ABB RAPID module: etna.mod

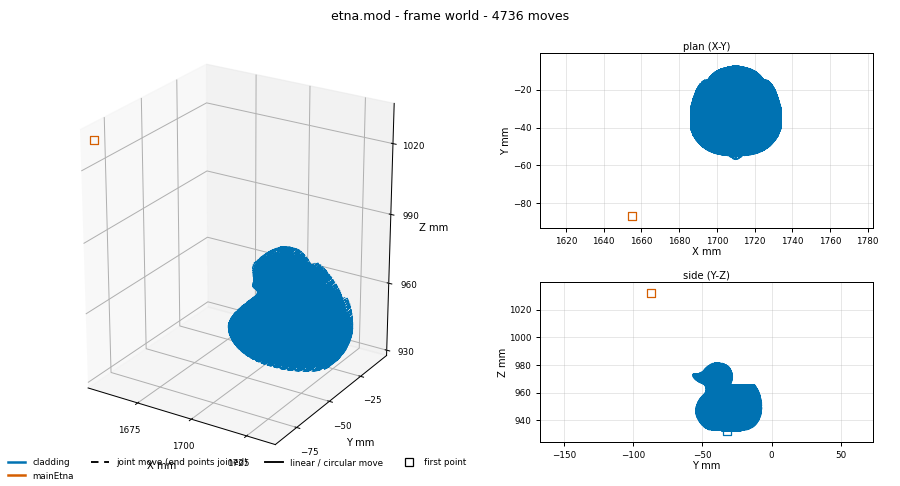
[picture p0: tool path of etna.mod in frame world, 4736 of 4736 moves have a stored position in this frame; points joined in program order, loops and branches not executed]
MODULE Etna

    PERS tooldata toolEtna:=[TRUE,[[530.0,46.8,126.6],[0.707107,0.000000,0.707107,0.000000]],[20,[70,30,123.5],[0,0,1,0],1,0,1]];
    PERS wobjdata wobjEtna:=[FALSE,TRUE,"",[[1655.0,-87.0,932.0],[1.000000,0.000000,0.000000,0.000000]],[[0,0,0],[1,0,0,0]]];

    VAR triggdata laserON;
    VAR triggdata laserOFF;

    CONST speeddata vl:=[8,500,5000,1000];


    CONST robtarget T0:=[[45.230797,54.660942,0.249511],[1.000000,0.000000,0.000000,0.000000],[0,0,-1,0],[9E+09,9E+09,9E+09,9E+09,9E+09,9E+09]];
    CONST robtarget T1:=[[45.230797,61.238206,0.249511],[1.000000,0.000000,0.000000,0.000000],[0,0,-1,0],[9E+09,9E+09,9E+09,9E+09,9E+09,9E+09]];
    CONST robtarget T2:=[[45.230797,54.660942,0.249511],[1.000000,0.000000,0.000000,0.000000],[0,0,-1,0],[9E+09,9E+09,9E+09,9E+09,9E+09,9E+09]];
    CONST robtarget T3:=[[45.230797,61.238206,0.249511],[1.000000,0.000000,0.000000,0.000000],[0,0,-1,0],[9E+09,9E+09,9E+09,9E+09,9E+09,9E+09]];
    CONST robtarget T4:=[[46.730803,63.450242,0.249511],[1.000000,0.000000,0.000000,0.000000],[0,0,-1,0],[9E+09,9E+09,9E+09,9E+09,9E+09,9E+09]];
    CONST robtarget T5:=[[46.730803,53.147305,0.249511],[1.000000,0.000000,0.000000,0.000000],[0,0,-1,0],[9E+09,9E+09,9E+09,9E+09,9E+09,9E+09]];
    CONST robtarget T6:=[[48.230809,51.823648,0.249511],[1.000000,0.000000,0.000000,0.000000],[0,0,-1,0],[9E+09,9E+09,9E+09,9E+09,9E+09,9E+09]];
    CONST robtarget T7:=[[48.230809,64.177413,0.249511],[1.000000,0.000000,0.000000,0.000000],[0,0,-1,0],[9E+09,9E+09,9E+09,9E+09,9E+09,9E+09]];
    CONST robtarget T8:=[[49.730815,64.861657,0.249511],[1.000000,0.000000,0.000000,0.000000],[0,0,-1,0],[9E+09,9E+09,9E+09,9E+09,9E+09,9E+09]];
    CONST robtarget T9:=[[49.730815,50.871953,0.249511],[1.000000,0.000000,0.000000,0.000000],[0,0,-1,0],[9E+09,9E+09,9E+09,9E+09,9E+09,9E+09]];
    CONST robtarget T10:=[[51.230821,50.942602,0.249511],[1.000000,0.000000,0.000000,0.000000],[0,0,-1,0],[9E+09,9E+09,9E+09,9E+09,9E+09,9E+09]];
    CONST robtarget T11:=[[51.230821,64.963902,0.249511],[1.000000,0.000000,0.000000,0.000000],[0,0,-1,0],[9E+09,9E+09,9E+09,9E+09,9E+09,9E+09]];
    CONST robtarget T12:=[[52.730827,64.937092,0.249511],[1.000000,0.000000,0.000000,0.000000],[0,0,-1,0],[9E+09,9E+09,9E+09,9E+09,9E+09,9E+09]];
    CONST robtarget T13:=[[52.730827,51.126270,0.249511],[1.000000,0.000000,0.000000,0.000000],[0,0,-1,0],[9E+09,9E+09,9E+09,9E+09,9E+09,9E+09]];
    CONST robtarget T14:=[[54.230833,51.704495,0.249511],[1.000000,0.000000,0.000000,0.000000],[0,0,-1,0],[9E+09,9E+09,9E+09,9E+09,9E+09,9E+09]];
    CONST robtarget T15:=[[54.230833,64.614973,0.249511],[1.000000,0.000000,0.000000,0.000000],[0,0,-1,0],[9E+09,9E+09,9E+09,9E+09,9E+09,9E+09]];
    CONST robtarget T16:=[[55.730839,64.604426,0.249511],[1.000000,0.000000,0.000000,0.000000],[0,0,-1,0],[9E+09,9E+09,9E+09,9E+09,9E+09,9E+09]];
    CONST robtarget T17:=[[55.730839,51.719275,0.249511],[1.000000,0.000000,0.000000,0.000000],[0,0,-1,0],[9E+09,9E+09,9E+09,9E+09,9E+09,9E+09]];
    CONST robtarget T18:=[[57.230845,51.141050,0.249511],[1.000000,0.000000,0.000000,0.000000],[0,0,-1,0],[9E+09,9E+09,9E+09,9E+09,9E+09,9E+09]];
    CONST robtarget T19:=[[57.230845,64.921597,0.249511],[1.000000,0.000000,0.000000,0.000000],[0,0,-1,0],[9E+09,9E+09,9E+09,9E+09,9E+09,9E+09]];
    CONST robtarget T20:=[[58.730851,64.951383,0.249511],[1.000000,0.000000,0.000000,0.000000],[0,0,-1,0],[9E+09,9E+09,9E+09,9E+09,9E+09,9E+09]];
    CONST robtarget T21:=[[58.730851,50.944648,0.249511],[1.000000,0.000000,0.000000,0.000000],[0,0,-1,0],[9E+09,9E+09,9E+09,9E+09,9E+09,9E+09]];
    CONST robtarget T22:=[[60.230857,50.873711,0.249511],[1.000000,0.000000,0.000000,0.000000],[0,0,-1,0],[9E+09,9E+09,9E+09,9E+09,9E+09,9E+09]];
    CONST robtarget T23:=[[60.230857,64.864853,0.249511],[1.000000,0.000000,0.000000,0.000000],[0,0,-1,0],[9E+09,9E+09,9E+09,9E+09,9E+09,9E+09]];
    CONST robtarget T24:=[[61.730863,64.173309,0.249511],[1.000000,0.000000,0.000000,0.000000],[0,0,-1,0],[9E+09,9E+09,9E+09,9E+09,9E+09,9E+09]];
    CONST robtarget T25:=[[61.730863,51.793503,0.249511],[1.000000,0.000000,0.000000,0.000000],[0,0,-1,0],[9E+09,9E+09,9E+09,9E+09,9E+09,9E+09]];
    CONST robtarget T26:=[[63.230869,53.117219,0.249511],[1.000000,0.000000,0.000000,0.000000],[0,0,-1,0],[9E+09,9E+09,9E+09,9E+09,9E+09,9E+09]];
    CONST robtarget T27:=[[63.230869,63.436121,0.249511],[1.000000,0.000000,0.000000,0.000000],[0,0,-1,0],[9E+09,9E+09,9E+09,9E+09,9E+09,9E+09]];
    CONST robtarget T28:=[[64.730875,61.202460,0.249511],[1.000000,0.000000,0.000000,0.000000],[0,0,-1,0],[9E+09,9E+09,9E+09,9E+09,9E+09,9E+09]];
    CONST robtarget T29:=[[64.730875,54.600120,0.249511],[1.000000,0.000000,0.000000,0.000000],[0,0,-1,0],[9E+09,9E+09,9E+09,9E+09,9E+09,9E+09]];
    CONST robtarget T30:=[[69.247273,52.344904,0.749521],[1.000000,0.000000,0.000000,0.000000],[0,0,-1,0],[9E+09,9E+09,9E+09,9E+09,9E+09,9E+09]];
    CONST robtarget T31:=[[69.247273,59.666876,0.749521],[1.000000,0.000000,0.000000,0.000000],[0,0,-1,0],[9E+09,9E+09,9E+09,9E+09,9E+09,9E+09]];
    CONST robtarget T32:=[[69.247273,52.344904,0.749521],[1.000000,0.000000,0.000000,0.000000],[0,0,-1,0],[9E+09,9E+09,9E+09,9E+09,9E+09,9E+09]];
    CONST robtarget T33:=[[69.247273,59.666876,0.749521],[1.000000,0.000000,0.000000,0.000000],[0,0,-1,0],[9E+09,9E+09,9E+09,9E+09,9E+09,9E+09]];
    CONST robtarget T34:=[[67.747267,63.988813,0.749521],[1.000000,0.000000,0.000000,0.000000],[0,0,-1,0],[9E+09,9E+09,9E+09,9E+09,9E+09,9E+09]];
    CONST robtarget T35:=[[67.747267,49.645310,0.749521],[1.000000,0.000000,0.000000,0.000000],[0,0,-1,0],[9E+09,9E+09,9E+09,9E+09,9E+09,9E+09]];
    CONST robtarget T36:=[[66.247261,47.604168,0.749521],[1.000000,0.000000,0.000000,0.000000],[0,0,-1,0],[9E+09,9E+09,9E+09,9E+09,9E+09,9E+09]];
    CONST robtarget T37:=[[66.247261,65.568560,0.749521],[1.000000,0.000000,0.000000,0.000000],[0,0,-1,0],[9E+09,9E+09,9E+09,9E+09,9E+09,9E+09]];
    CONST robtarget T38:=[[64.747255,66.220066,0.749521],[1.000000,0.000000,0.000000,0.000000],[0,0,-1,0],[9E+09,9E+09,9E+09,9E+09,9E+09,9E+09]];
    CONST robtarget T39:=[[64.747255,46.247530,0.749521],[1.000000,0.000000,0.000000,0.000000],[0,0,-1,0],[9E+09,9E+09,9E+09,9E+09,9E+09,9E+09]];
    CONST robtarget T40:=[[63.247249,45.205197,0.749521],[1.000000,0.000000,0.000000,0.000000],[0,0,-1,0],[9E+09,9E+09,9E+09,9E+09,9E+09,9E+09]];
    CONST robtarget T41:=[[63.247249,66.893237,0.749521],[1.000000,0.000000,0.000000,0.000000],[0,0,-1,0],[9E+09,9E+09,9E+09,9E+09,9E+09,9E+09]];
    CONST robtarget T42:=[[61.747243,67.230044,0.749521],[1.000000,0.000000,0.000000,0.000000],[0,0,-1,0],[9E+09,9E+09,9E+09,9E+09,9E+09,9E+09]];
    CONST robtarget T43:=[[61.747243,44.353778,0.749521],[1.000000,0.000000,0.000000,0.000000],[0,0,-1,0],[9E+09,9E+09,9E+09,9E+09,9E+09,9E+09]];
    CONST robtarget T44:=[[60.247237,43.858747,0.749521],[1.000000,0.000000,0.000000,0.000000],[0,0,-1,0],[9E+09,9E+09,9E+09,9E+09,9E+09,9E+09]];
    CONST robtarget T45:=[[60.247237,67.502036,0.749521],[1.000000,0.000000,0.000000,0.000000],[0,0,-1,0],[9E+09,9E+09,9E+09,9E+09,9E+09,9E+09]];
    CONST robtarget T46:=[[58.747231,67.649975,0.749521],[1.000000,0.000000,0.000000,0.000000],[0,0,-1,0],[9E+09,9E+09,9E+09,9E+09,9E+09,9E+09]];
    CONST robtarget T47:=[[58.747231,43.776283,0.749521],[1.000000,0.000000,0.000000,0.000000],[0,0,-1,0],[9E+09,9E+09,9E+09,9E+09,9E+09,9E+09]];
    CONST robtarget T48:=[[57.247225,43.725602,0.749521],[1.000000,0.000000,0.000000,0.000000],[0,0,-1,0],[9E+09,9E+09,9E+09,9E+09,9E+09,9E+09]];
    CONST robtarget T49:=[[57.247225,67.674292,0.749521],[1.000000,0.000000,0.000000,0.000000],[0,0,-1,0],[9E+09,9E+09,9E+09,9E+09,9E+09,9E+09]];
    CONST robtarget T50:=[[55.747219,67.566917,0.749521],[1.000000,0.000000,0.000000,0.000000],[0,0,-1,0],[9E+09,9E+09,9E+09,9E+09,9E+09,9E+09]];
    CONST robtarget T51:=[[55.747219,43.852921,0.749521],[1.000000,0.000000,0.000000,0.000000],[0,0,-1,0],[9E+09,9E+09,9E+09,9E+09,9E+09,9E+09]];
    CONST robtarget T52:=[[54.247213,43.852451,0.749521],[1.000000,0.000000,0.000000,0.000000],[0,0,-1,0],[9E+09,9E+09,9E+09,9E+09,9E+09,9E+09]];
    CONST robtarget T53:=[[54.247213,67.567771,0.749521],[1.000000,0.000000,0.000000,0.000000],[0,0,-1,0],[9E+09,9E+09,9E+09,9E+09,9E+09,9E+09]];
    CONST robtarget T54:=[[52.747207,67.674435,0.749521],[1.000000,0.000000,0.000000,0.000000],[0,0,-1,0],[9E+09,9E+09,9E+09,9E+09,9E+09,9E+09]];
    CONST robtarget T55:=[[52.747207,43.725093,0.749521],[1.000000,0.000000,0.000000,0.000000],[0,0,-1,0],[9E+09,9E+09,9E+09,9E+09,9E+09,9E+09]];
    CONST robtarget T56:=[[51.247201,43.776532,0.749521],[1.000000,0.000000,0.000000,0.000000],[0,0,-1,0],[9E+09,9E+09,9E+09,9E+09,9E+09,9E+09]];
    CONST robtarget T57:=[[51.247201,67.650171,0.749521],[1.000000,0.000000,0.000000,0.000000],[0,0,-1,0],[9E+09,9E+09,9E+09,9E+09,9E+09,9E+09]];
    CONST robtarget T58:=[[49.747195,67.501890,0.749521],[1.000000,0.000000,0.000000,0.000000],[0,0,-1,0],[9E+09,9E+09,9E+09,9E+09,9E+09,9E+09]];
    CONST robtarget T59:=[[49.747195,43.860589,0.749521],[1.000000,0.000000,0.000000,0.000000],[0,0,-1,0],[9E+09,9E+09,9E+09,9E+09,9E+09,9E+09]];
    CONST robtarget T60:=[[48.247189,44.355622,0.749521],[1.000000,0.000000,0.000000,0.000000],[0,0,-1,0],[9E+09,9E+09,9E+09,9E+09,9E+09,9E+09]];
    CONST robtarget T61:=[[48.247189,67.230329,0.749521],[1.000000,0.000000,0.000000,0.000000],[0,0,-1,0],[9E+09,9E+09,9E+09,9E+09,9E+09,9E+09]];
    CONST robtarget T62:=[[46.747183,66.892498,0.749521],[1.000000,0.000000,0.000000,0.000000],[0,0,-1,0],[9E+09,9E+09,9E+09,9E+09,9E+09,9E+09]];
    CONST robtarget T63:=[[46.747183,45.207884,0.749521],[1.000000,0.000000,0.000000,0.000000],[0,0,-1,0],[9E+09,9E+09,9E+09,9E+09,9E+09,9E+09]];
    CONST robtarget T64:=[[45.247177,46.252109,0.749521],[1.000000,0.000000,0.000000,0.000000],[0,0,-1,0],[9E+09,9E+09,9E+09,9E+09,9E+09,9E+09]];
    CONST robtarget T65:=[[45.247177,66.220428,0.749521],[1.000000,0.000000,0.000000,0.000000],[0,0,-1,0],[9E+09,9E+09,9E+09,9E+09,9E+09,9E+09]];
    CONST robtarget T66:=[[43.747171,65.569397,0.749521],[1.000000,0.000000,0.000000,0.000000],[0,0,-1,0],[9E+09,9E+09,9E+09,9E+09,9E+09,9E+09]];
    CONST robtarget T67:=[[43.747171,47.613223,0.749521],[1.000000,0.000000,0.000000,0.000000],[0,0,-1,0],[9E+09,9E+09,9E+09,9E+09,9E+09,9E+09]];
    CONST robtarget T68:=[[42.247165,49.652254,0.749521],[1.000000,0.000000,0.000000,0.000000],[0,0,-1,0],[9E+09,9E+09,9E+09,9E+09,9E+09,9E+09]];
    CONST robtarget T69:=[[42.247165,63.997482,0.749521],[1.000000,0.000000,0.000000,0.000000],[0,0,-1,0],[9E+09,9E+09,9E+09,9E+09,9E+09,9E+09]];
    CONST robtarget T70:=[[40.747159,59.721737,0.749521],[1.000000,0.000000,0.000000,0.000000],[0,0,-1,0],[9E+09,9E+09,9E+09,9E+09,9E+09,9E+09]];
    CONST robtarget T71:=[[40.747159,52.382179,0.749521],[1.000000,0.000000,0.000000,0.000000],[0,0,-1,0],[9E+09,9E+09,9E+09,9E+09,9E+09,9E+09]];
    CONST robtarget T72:=[[38.499544,50.308177,1.249531],[1.000000,0.000000,0.000000,0.000000],[0,0,-1,0],[9E+09,9E+09,9E+09,9E+09,9E+09,9E+09]];
    CONST robtarget T73:=[[38.499544,60.298450,1.249531],[1.000000,0.000000,0.000000,0.000000],[0,0,-1,0],[9E+09,9E+09,9E+09,9E+09,9E+09,9E+09]];
    CONST robtarget T74:=[[38.499544,50.308177,1.249531],[1.000000,0.000000,0.000000,0.000000],[0,0,-1,0],[9E+09,9E+09,9E+09,9E+09,9E+09,9E+09]];
    CONST robtarget T75:=[[38.499544,60.298450,1.249531],[1.000000,0.000000,0.000000,0.000000],[0,0,-1,0],[9E+09,9E+09,9E+09,9E+09,9E+09,9E+09]];
    CONST robtarget T76:=[[39.999550,64.489479,1.249531],[1.000000,0.000000,0.000000,0.000000],[0,0,-1,0],[9E+09,9E+09,9E+09,9E+09,9E+09,9E+09]];
    CONST robtarget T77:=[[39.999550,47.499380,1.249531],[1.000000,0.000000,0.000000,0.000000],[0,0,-1,0],[9E+09,9E+09,9E+09,9E+09,9E+09,9E+09]];
    CONST robtarget T78:=[[41.499556,46.077025,1.249531],[1.000000,0.000000,0.000000,0.000000],[0,0,-1,0],[9E+09,9E+09,9E+09,9E+09,9E+09,9E+09]];
    CONST robtarget T79:=[[41.499556,66.064956,1.249531],[1.000000,0.000000,0.000000,0.000000],[0,0,-1,0],[9E+09,9E+09,9E+09,9E+09,9E+09,9E+09]];
    CONST robtarget T80:=[[42.999562,67.172158,1.249531],[1.000000,0.000000,0.000000,0.000000],[0,0,-1,0],[9E+09,9E+09,9E+09,9E+09,9E+09,9E+09]];
    CONST robtarget T81:=[[42.999562,44.769816,1.249531],[1.000000,0.000000,0.000000,0.000000],[0,0,-1,0],[9E+09,9E+09,9E+09,9E+09,9E+09,9E+09]];
    CONST robtarget T82:=[[44.499568,44.074901,1.249531],[1.000000,0.000000,0.000000,0.000000],[0,0,-1,0],[9E+09,9E+09,9E+09,9E+09,9E+09,9E+09]];
    CONST robtarget T83:=[[44.499568,68.035223,1.249531],[1.000000,0.000000,0.000000,0.000000],[0,0,-1,0],[9E+09,9E+09,9E+09,9E+09,9E+09,9E+09]];
    CONST robtarget T84:=[[45.999574,68.487089,1.249531],[1.000000,0.000000,0.000000,0.000000],[0,0,-1,0],[9E+09,9E+09,9E+09,9E+09,9E+09,9E+09]];
    CONST robtarget T85:=[[45.999574,43.291383,1.249531],[1.000000,0.000000,0.000000,0.000000],[0,0,-1,0],[9E+09,9E+09,9E+09,9E+09,9E+09,9E+09]];
    CONST robtarget T86:=[[47.499580,42.569706,1.249531],[1.000000,0.000000,0.000000,0.000000],[0,0,-1,0],[9E+09,9E+09,9E+09,9E+09,9E+09,9E+09]];
    CONST robtarget T87:=[[47.499580,68.938955,1.249531],[1.000000,0.000000,0.000000,0.000000],[0,0,-1,0],[9E+09,9E+09,9E+09,9E+09,9E+09,9E+09]];
    CONST robtarget T88:=[[48.999586,69.156373,1.249531],[1.000000,0.000000,0.000000,0.000000],[0,0,-1,0],[9E+09,9E+09,9E+09,9E+09,9E+09,9E+09]];
    CONST robtarget T89:=[[48.999586,42.028761,1.249531],[1.000000,0.000000,0.000000,0.000000],[0,0,-1,0],[9E+09,9E+09,9E+09,9E+09,9E+09,9E+09]];
    CONST robtarget T90:=[[50.499592,41.629502,1.249531],[1.000000,0.000000,0.000000,0.000000],[0,0,-1,0],[9E+09,9E+09,9E+09,9E+09,9E+09,9E+09]];
    CONST robtarget T91:=[[50.499592,69.313504,1.249531],[1.000000,0.000000,0.000000,0.000000],[0,0,-1,0],[9E+09,9E+09,9E+09,9E+09,9E+09,9E+09]];
    CONST robtarget T92:=[[51.999598,69.380595,1.249531],[1.000000,0.000000,0.000000,0.000000],[0,0,-1,0],[9E+09,9E+09,9E+09,9E+09,9E+09,9E+09]];
    CONST robtarget T93:=[[51.999598,41.543714,1.249531],[1.000000,0.000000,0.000000,0.000000],[0,0,-1,0],[9E+09,9E+09,9E+09,9E+09,9E+09,9E+09]];
    CONST robtarget T94:=[[53.499604,41.519114,1.249531],[1.000000,0.000000,0.000000,0.000000],[0,0,-1,0],[9E+09,9E+09,9E+09,9E+09,9E+09,9E+09]];
    CONST robtarget T95:=[[53.499604,69.370940,1.249531],[1.000000,0.000000,0.000000,0.000000],[0,0,-1,0],[9E+09,9E+09,9E+09,9E+09,9E+09,9E+09]];
    CONST robtarget T96:=[[54.999610,69.325352,1.249531],[1.000000,0.000000,0.000000,0.000000],[0,0,-1,0],[9E+09,9E+09,9E+09,9E+09,9E+09,9E+09]];
    CONST robtarget T97:=[[54.999610,41.622696,1.249531],[1.000000,0.000000,0.000000,0.000000],[0,0,-1,0],[9E+09,9E+09,9E+09,9E+09,9E+09,9E+09]];
    CONST robtarget T98:=[[56.499616,41.519131,1.249531],[1.000000,0.000000,0.000000,0.000000],[0,0,-1,0],[9E+09,9E+09,9E+09,9E+09,9E+09,9E+09]];
    CONST robtarget T99:=[[56.499616,69.370908,1.249531],[1.000000,0.000000,0.000000,0.000000],[0,0,-1,0],[9E+09,9E+09,9E+09,9E+09,9E+09,9E+09]];
    CONST robtarget T100:=[[57.999622,69.380616,1.249531],[1.000000,0.000000,0.000000,0.000000],[0,0,-1,0],[9E+09,9E+09,9E+09,9E+09,9E+09,9E+09]];
    CONST robtarget T101:=[[57.999622,41.543669,1.249531],[1.000000,0.000000,0.000000,0.000000],[0,0,-1,0],[9E+09,9E+09,9E+09,9E+09,9E+09,9E+09]];
    CONST robtarget T102:=[[59.499628,41.629457,1.249531],[1.000000,0.000000,0.000000,0.000000],[0,0,-1,0],[9E+09,9E+09,9E+09,9E+09,9E+09,9E+09]];
    CONST robtarget T103:=[[59.499628,69.313582,1.249531],[1.000000,0.000000,0.000000,0.000000],[0,0,-1,0],[9E+09,9E+09,9E+09,9E+09,9E+09,9E+09]];
    CONST robtarget T104:=[[60.999634,69.156474,1.249531],[1.000000,0.000000,0.000000,0.000000],[0,0,-1,0],[9E+09,9E+09,9E+09,9E+09,9E+09,9E+09]];
    CONST robtarget T105:=[[60.999634,42.028474,1.249531],[1.000000,0.000000,0.000000,0.000000],[0,0,-1,0],[9E+09,9E+09,9E+09,9E+09,9E+09,9E+09]];
    CONST robtarget T106:=[[62.499640,42.569419,1.249531],[1.000000,0.000000,0.000000,0.000000],[0,0,-1,0],[9E+09,9E+09,9E+09,9E+09,9E+09,9E+09]];
    CONST robtarget T107:=[[62.499640,68.939194,1.249531],[1.000000,0.000000,0.000000,0.000000],[0,0,-1,0],[9E+09,9E+09,9E+09,9E+09,9E+09,9E+09]];
    CONST robtarget T108:=[[63.999646,68.487328,1.249531],[1.000000,0.000000,0.000000,0.000000],[0,0,-1,0],[9E+09,9E+09,9E+09,9E+09,9E+09,9E+09]];
    CONST robtarget T109:=[[63.999646,43.290925,1.249531],[1.000000,0.000000,0.000000,0.000000],[0,0,-1,0],[9E+09,9E+09,9E+09,9E+09,9E+09,9E+09]];
    CONST robtarget T110:=[[65.499652,44.074529,1.249531],[1.000000,0.000000,0.000000,0.000000],[0,0,-1,0],[9E+09,9E+09,9E+09,9E+09,9E+09,9E+09]];
    CONST robtarget T111:=[[65.499652,68.035462,1.249531],[1.000000,0.000000,0.000000,0.000000],[0,0,-1,0],[9E+09,9E+09,9E+09,9E+09,9E+09,9E+09]];
    CONST robtarget T112:=[[66.999658,67.172468,1.249531],[1.000000,0.000000,0.000000,0.000000],[0,0,-1,0],[9E+09,9E+09,9E+09,9E+09,9E+09,9E+09]];
    CONST robtarget T113:=[[66.999658,44.769447,1.249531],[1.000000,0.000000,0.000000,0.000000],[0,0,-1,0],[9E+09,9E+09,9E+09,9E+09,9E+09,9E+09]];
    CONST robtarget T114:=[[68.499664,46.076202,1.249531],[1.000000,0.000000,0.000000,0.000000],[0,0,-1,0],[9E+09,9E+09,9E+09,9E+09,9E+09,9E+09]];
    CONST robtarget T115:=[[68.499664,66.065017,1.249531],[1.000000,0.000000,0.000000,0.000000],[0,0,-1,0],[9E+09,9E+09,9E+09,9E+09,9E+09,9E+09]];
    CONST robtarget T116:=[[69.999670,64.488299,1.249531],[1.000000,0.000000,0.000000,0.000000],[0,0,-1,0],[9E+09,9E+09,9E+09,9E+09,9E+09,9E+09]];
    CONST robtarget T117:=[[69.999670,47.498673,1.249531],[1.000000,0.000000,0.000000,0.000000],[0,0,-1,0],[9E+09,9E+09,9E+09,9E+09,9E+09,9E+09]];
    CONST robtarget T118:=[[71.499676,50.306050,1.249531],[1.000000,0.000000,0.000000,0.000000],[0,0,-1,0],[9E+09,9E+09,9E+09,9E+09,9E+09,9E+09]];
    CONST robtarget T119:=[[71.499676,60.263678,1.249531],[1.000000,0.000000,0.000000,0.000000],[0,0,-1,0],[9E+09,9E+09,9E+09,9E+09,9E+09,9E+09]];
    CONST robtarget T120:=[[73.000077,49.540950,1.749541],[1.000000,0.000000,0.000000,0.000000],[0,0,-1,0],[9E+09,9E+09,9E+09,9E+09,9E+09,9E+09]];
    CONST robtarget T121:=[[73.000077,58.164737,1.749541],[1.000000,0.000000,0.000000,0.000000],[0,0,-1,0],[9E+09,9E+09,9E+09,9E+09,9E+09,9E+09]];
    CONST robtarget T122:=[[73.000077,49.540950,1.749541],[1.000000,0.000000,0.000000,0.000000],[0,0,-1,0],[9E+09,9E+09,9E+09,9E+09,9E+09,9E+09]];
    CONST robtarget T123:=[[73.000077,58.164737,1.749541],[1.000000,0.000000,0.000000,0.000000],[0,0,-1,0],[9E+09,9E+09,9E+09,9E+09,9E+09,9E+09]];
    CONST robtarget T124:=[[71.500071,63.783623,1.749541],[1.000000,0.000000,0.000000,0.000000],[0,0,-1,0],[9E+09,9E+09,9E+09,9E+09,9E+09,9E+09]];
    CONST robtarget T125:=[[71.500071,46.656280,1.749541],[1.000000,0.000000,0.000000,0.000000],[0,0,-1,0],[9E+09,9E+09,9E+09,9E+09,9E+09,9E+09]];
    CONST robtarget T126:=[[70.000065,45.101701,1.749541],[1.000000,0.000000,0.000000,0.000000],[0,0,-1,0],[9E+09,9E+09,9E+09,9E+09,9E+09,9E+09]];
    CONST robtarget T127:=[[70.000065,66.271272,1.749541],[1.000000,0.000000,0.000000,0.000000],[0,0,-1,0],[9E+09,9E+09,9E+09,9E+09,9E+09,9E+09]];
    CONST robtarget T128:=[[68.500059,67.688442,1.749541],[1.000000,0.000000,0.000000,0.000000],[0,0,-1,0],[9E+09,9E+09,9E+09,9E+09,9E+09,9E+09]];
    CONST robtarget T129:=[[68.500059,44.151934,1.749541],[1.000000,0.000000,0.000000,0.000000],[0,0,-1,0],[9E+09,9E+09,9E+09,9E+09,9E+09,9E+09]];
    CONST robtarget T130:=[[67.000053,43.202167,1.749541],[1.000000,0.000000,0.000000,0.000000],[0,0,-1,0],[9E+09,9E+09,9E+09,9E+09,9E+09,9E+09]];
    CONST robtarget T131:=[[67.000053,68.457961,1.749541],[1.000000,0.000000,0.000000,0.000000],[0,0,-1,0],[9E+09,9E+09,9E+09,9E+09,9E+09,9E+09]];
    CONST robtarget T132:=[[65.500047,69.385771,1.749541],[1.000000,0.000000,0.000000,0.000000],[0,0,-1,0],[9E+09,9E+09,9E+09,9E+09,9E+09,9E+09]];
    CONST robtarget T133:=[[65.500047,42.445663,1.749541],[1.000000,0.000000,0.000000,0.000000],[0,0,-1,0],[9E+09,9E+09,9E+09,9E+09,9E+09,9E+09]];
    CONST robtarget T134:=[[64.000041,41.874691,1.749541],[1.000000,0.000000,0.000000,0.000000],[0,0,-1,0],[9E+09,9E+09,9E+09,9E+09,9E+09,9E+09]];
    CONST robtarget T135:=[[64.000041,69.938803,1.749541],[1.000000,0.000000,0.000000,0.000000],[0,0,-1,0],[9E+09,9E+09,9E+09,9E+09,9E+09,9E+09]];
    CONST robtarget T136:=[[62.500035,70.380115,1.749541],[1.000000,0.000000,0.000000,0.000000],[0,0,-1,0],[9E+09,9E+09,9E+09,9E+09,9E+09,9E+09]];
    CONST robtarget T137:=[[62.500035,41.341429,1.749541],[1.000000,0.000000,0.000000,0.000000],[0,0,-1,0],[9E+09,9E+09,9E+09,9E+09,9E+09,9E+09]];
    CONST robtarget T138:=[[61.000029,40.952491,1.749541],[1.000000,0.000000,0.000000,0.000000],[0,0,-1,0],[9E+09,9E+09,9E+09,9E+09,9E+09,9E+09]];
    CONST robtarget T139:=[[61.000029,70.613365,1.749541],[1.000000,0.000000,0.000000,0.000000],[0,0,-1,0],[9E+09,9E+09,9E+09,9E+09,9E+09,9E+09]];
    CONST robtarget T140:=[[59.500023,70.730845,1.749541],[1.000000,0.000000,0.000000,0.000000],[0,0,-1,0],[9E+09,9E+09,9E+09,9E+09,9E+09,9E+09]];
    CONST robtarget T141:=[[59.500023,40.606692,1.749541],[1.000000,0.000000,0.000000,0.000000],[0,0,-1,0],[9E+09,9E+09,9E+09,9E+09,9E+09,9E+09]];
    CONST robtarget T142:=[[58.000017,40.513780,1.749541],[1.000000,0.000000,0.000000,0.000000],[0,0,-1,0],[9E+09,9E+09,9E+09,9E+09,9E+09,9E+09]];
    CONST robtarget T143:=[[58.000017,70.803110,1.749541],[1.000000,0.000000,0.000000,0.000000],[0,0,-1,0],[9E+09,9E+09,9E+09,9E+09,9E+09,9E+09]];
    CONST robtarget T144:=[[56.500011,70.842486,1.749541],[1.000000,0.000000,0.000000,0.000000],[0,0,-1,0],[9E+09,9E+09,9E+09,9E+09,9E+09,9E+09]];
    CONST robtarget T145:=[[56.500011,40.485362,1.749541],[1.000000,0.000000,0.000000,0.000000],[0,0,-1,0],[9E+09,9E+09,9E+09,9E+09,9E+09,9E+09]];
    CONST robtarget T146:=[[55.000005,40.512783,1.749541],[1.000000,0.000000,0.000000,0.000000],[0,0,-1,0],[9E+09,9E+09,9E+09,9E+09,9E+09,9E+09]];
    CONST robtarget T147:=[[55.000005,70.830121,1.749541],[1.000000,0.000000,0.000000,0.000000],[0,0,-1,0],[9E+09,9E+09,9E+09,9E+09,9E+09,9E+09]];
    CONST robtarget T148:=[[53.499999,70.842488,1.749541],[1.000000,0.000000,0.000000,0.000000],[0,0,-1,0],[9E+09,9E+09,9E+09,9E+09,9E+09,9E+09]];
    CONST robtarget T149:=[[53.499999,40.485362,1.749541],[1.000000,0.000000,0.000000,0.000000],[0,0,-1,0],[9E+09,9E+09,9E+09,9E+09,9E+09,9E+09]];
    CONST robtarget T150:=[[51.999993,40.513780,1.749541],[1.000000,0.000000,0.000000,0.000000],[0,0,-1,0],[9E+09,9E+09,9E+09,9E+09,9E+09,9E+09]];
    CONST robtarget T151:=[[51.999993,70.803110,1.749541],[1.000000,0.000000,0.000000,0.000000],[0,0,-1,0],[9E+09,9E+09,9E+09,9E+09,9E+09,9E+09]];
    CONST robtarget T152:=[[50.499987,70.730845,1.749541],[1.000000,0.000000,0.000000,0.000000],[0,0,-1,0],[9E+09,9E+09,9E+09,9E+09,9E+09,9E+09]];
    CONST robtarget T153:=[[50.499987,40.606692,1.749541],[1.000000,0.000000,0.000000,0.000000],[0,0,-1,0],[9E+09,9E+09,9E+09,9E+09,9E+09,9E+09]];
    CONST robtarget T154:=[[48.999981,40.952493,1.749541],[1.000000,0.000000,0.000000,0.000000],[0,0,-1,0],[9E+09,9E+09,9E+09,9E+09,9E+09,9E+09]];
    CONST robtarget T155:=[[48.999981,70.613365,1.749541],[1.000000,0.000000,0.000000,0.000000],[0,0,-1,0],[9E+09,9E+09,9E+09,9E+09,9E+09,9E+09]];
    CONST robtarget T156:=[[47.499975,70.380114,1.749541],[1.000000,0.000000,0.000000,0.000000],[0,0,-1,0],[9E+09,9E+09,9E+09,9E+09,9E+09,9E+09]];
    CONST robtarget T157:=[[47.499975,41.341430,1.749541],[1.000000,0.000000,0.000000,0.000000],[0,0,-1,0],[9E+09,9E+09,9E+09,9E+09,9E+09,9E+09]];
    CONST robtarget T158:=[[45.999969,41.874694,1.749541],[1.000000,0.000000,0.000000,0.000000],[0,0,-1,0],[9E+09,9E+09,9E+09,9E+09,9E+09,9E+09]];
    CONST robtarget T159:=[[45.999969,69.938801,1.749541],[1.000000,0.000000,0.000000,0.000000],[0,0,-1,0],[9E+09,9E+09,9E+09,9E+09,9E+09,9E+09]];
    CONST robtarget T160:=[[44.499963,69.385768,1.749541],[1.000000,0.000000,0.000000,0.000000],[0,0,-1,0],[9E+09,9E+09,9E+09,9E+09,9E+09,9E+09]];
    CONST robtarget T161:=[[44.499963,42.445669,1.749541],[1.000000,0.000000,0.000000,0.000000],[0,0,-1,0],[9E+09,9E+09,9E+09,9E+09,9E+09,9E+09]];
    CONST robtarget T162:=[[42.999957,43.202177,1.749541],[1.000000,0.000000,0.000000,0.000000],[0,0,-1,0],[9E+09,9E+09,9E+09,9E+09,9E+09,9E+09]];
    CONST robtarget T163:=[[42.999957,68.457958,1.749541],[1.000000,0.000000,0.000000,0.000000],[0,0,-1,0],[9E+09,9E+09,9E+09,9E+09,9E+09,9E+09]];
    CONST robtarget T164:=[[41.499951,67.688441,1.749541],[1.000000,0.000000,0.000000,0.000000],[0,0,-1,0],[9E+09,9E+09,9E+09,9E+09,9E+09,9E+09]];
    CONST robtarget T165:=[[41.499951,44.151941,1.749541],[1.000000,0.000000,0.000000,0.000000],[0,0,-1,0],[9E+09,9E+09,9E+09,9E+09,9E+09,9E+09]];
    CONST robtarget T166:=[[39.999945,45.101704,1.749541],[1.000000,0.000000,0.000000,0.000000],[0,0,-1,0],[9E+09,9E+09,9E+09,9E+09,9E+09,9E+09]];
    CONST robtarget T167:=[[39.999945,66.272627,1.749541],[1.000000,0.000000,0.000000,0.000000],[0,0,-1,0],[9E+09,9E+09,9E+09,9E+09,9E+09,9E+09]];
    CONST robtarget T168:=[[38.499939,63.788624,1.749541],[1.000000,0.000000,0.000000,0.000000],[0,0,-1,0],[9E+09,9E+09,9E+09,9E+09,9E+09,9E+09]];
    CONST robtarget T169:=[[38.499939,46.656285,1.749541],[1.000000,0.000000,0.000000,0.000000],[0,0,-1,0],[9E+09,9E+09,9E+09,9E+09,9E+09,9E+09]];
    CONST robtarget T170:=[[36.999933,49.540961,1.749541],[1.000000,0.000000,0.000000,0.000000],[0,0,-1,0],[9E+09,9E+09,9E+09,9E+09,9E+09,9E+09]];
    CONST robtarget T171:=[[36.999933,58.175696,1.749541],[1.000000,0.000000,0.000000,0.000000],[0,0,-1,0],[9E+09,9E+09,9E+09,9E+09,9E+09,9E+09]];
    CONST robtarget T172:=[[36.250324,48.397228,2.249551],[1.000000,0.000000,0.000000,0.000000],[0,0,-1,0],[9E+09,9E+09,9E+09,9E+09,9E+09,9E+09]];
    CONST robtarget T173:=[[36.250324,59.214847,2.249551],[1.000000,0.000000,0.000000,0.000000],[0,0,-1,0],[9E+09,9E+09,9E+09,9E+09,9E+09,9E+09]];
    CONST robtarget T174:=[[36.250324,48.397228,2.249551],[1.000000,0.000000,0.000000,0.000000],[0,0,-1,0],[9E+09,9E+09,9E+09,9E+09,9E+09,9E+09]];
    CONST robtarget T175:=[[36.250324,59.214847,2.249551],[1.000000,0.000000,0.000000,0.000000],[0,0,-1,0],[9E+09,9E+09,9E+09,9E+09,9E+09,9E+09]];
    CONST robtarget T176:=[[37.750330,64.085193,2.249551],[1.000000,0.000000,0.000000,0.000000],[0,0,-1,0],[9E+09,9E+09,9E+09,9E+09,9E+09,9E+09]];
    CONST robtarget T177:=[[37.750330,45.991942,2.249551],[1.000000,0.000000,0.000000,0.000000],[0,0,-1,0],[9E+09,9E+09,9E+09,9E+09,9E+09,9E+09]];
    CONST robtarget T178:=[[39.250336,44.568903,2.249551],[1.000000,0.000000,0.000000,0.000000],[0,0,-1,0],[9E+09,9E+09,9E+09,9E+09,9E+09,9E+09]];
    CONST robtarget T179:=[[39.250336,66.308930,2.249551],[1.000000,0.000000,0.000000,0.000000],[0,0,-1,0],[9E+09,9E+09,9E+09,9E+09,9E+09,9E+09]];
    CONST robtarget T180:=[[40.750342,67.989973,2.249551],[1.000000,0.000000,0.000000,0.000000],[0,0,-1,0],[9E+09,9E+09,9E+09,9E+09,9E+09,9E+09]];
    CONST robtarget T181:=[[40.750342,43.327424,2.249551],[1.000000,0.000000,0.000000,0.000000],[0,0,-1,0],[9E+09,9E+09,9E+09,9E+09,9E+09,9E+09]];
    CONST robtarget T182:=[[42.250348,42.606898,2.249551],[1.000000,0.000000,0.000000,0.000000],[0,0,-1,0],[9E+09,9E+09,9E+09,9E+09,9E+09,9E+09]];
    CONST robtarget T183:=[[42.250348,69.121905,2.249551],[1.000000,0.000000,0.000000,0.000000],[0,0,-1,0],[9E+09,9E+09,9E+09,9E+09,9E+09,9E+09]];
    CONST robtarget T184:=[[43.750354,70.008448,2.249551],[1.000000,0.000000,0.000000,0.000000],[0,0,-1,0],[9E+09,9E+09,9E+09,9E+09,9E+09,9E+09]];
    CONST robtarget T185:=[[43.750354,41.846430,2.249551],[1.000000,0.000000,0.000000,0.000000],[0,0,-1,0],[9E+09,9E+09,9E+09,9E+09,9E+09,9E+09]];
    CONST robtarget T186:=[[45.250360,41.202387,2.249551],[1.000000,0.000000,0.000000,0.000000],[0,0,-1,0],[9E+09,9E+09,9E+09,9E+09,9E+09,9E+09]];
    CONST robtarget T187:=[[45.250360,70.831245,2.249551],[1.000000,0.000000,0.000000,0.000000],[0,0,-1,0],[9E+09,9E+09,9E+09,9E+09,9E+09,9E+09]];
    CONST robtarget T188:=[[46.750366,71.247041,2.249551],[1.000000,0.000000,0.000000,0.000000],[0,0,-1,0],[9E+09,9E+09,9E+09,9E+09,9E+09,9E+09]];
    CONST robtarget T189:=[[46.750366,40.618606,2.249551],[1.000000,0.000000,0.000000,0.000000],[0,0,-1,0],[9E+09,9E+09,9E+09,9E+09,9E+09,9E+09]];
    CONST robtarget T190:=[[48.250372,40.149877,2.249551],[1.000000,0.000000,0.000000,0.000000],[0,0,-1,0],[9E+09,9E+09,9E+09,9E+09,9E+09,9E+09]];
    CONST robtarget T191:=[[48.250372,71.629090,2.249551],[1.000000,0.000000,0.000000,0.000000],[0,0,-1,0],[9E+09,9E+09,9E+09,9E+09,9E+09,9E+09]];
    CONST robtarget T192:=[[49.750378,71.805464,2.249551],[1.000000,0.000000,0.000000,0.000000],[0,0,-1,0],[9E+09,9E+09,9E+09,9E+09,9E+09,9E+09]];
    CONST robtarget T193:=[[49.750378,39.761399,2.249551],[1.000000,0.000000,0.000000,0.000000],[0,0,-1,0],[9E+09,9E+09,9E+09,9E+09,9E+09,9E+09]];
    CONST robtarget T194:=[[51.250384,39.536943,2.249551],[1.000000,0.000000,0.000000,0.000000],[0,0,-1,0],[9E+09,9E+09,9E+09,9E+09,9E+09,9E+09]];
    CONST robtarget T195:=[[51.250384,71.906931,2.249551],[1.000000,0.000000,0.000000,0.000000],[0,0,-1,0],[9E+09,9E+09,9E+09,9E+09,9E+09,9E+09]];
    CONST robtarget T196:=[[52.750390,71.973450,2.249551],[1.000000,0.000000,0.000000,0.000000],[0,0,-1,0],[9E+09,9E+09,9E+09,9E+09,9E+09,9E+09]];
    CONST robtarget T197:=[[52.750390,39.440952,2.249551],[1.000000,0.000000,0.000000,0.000000],[0,0,-1,0],[9E+09,9E+09,9E+09,9E+09,9E+09,9E+09]];
    CONST robtarget T198:=[[54.250396,39.462104,2.249551],[1.000000,0.000000,0.000000,0.000000],[0,0,-1,0],[9E+09,9E+09,9E+09,9E+09,9E+09,9E+09]];
    CONST robtarget T199:=[[54.250396,72.010261,2.249551],[1.000000,0.000000,0.000000,0.000000],[0,0,-1,0],[9E+09,9E+09,9E+09,9E+09,9E+09,9E+09]];
    CONST robtarget T200:=[[55.750402,72.010251,2.249551],[1.000000,0.000000,0.000000,0.000000],[0,0,-1,0],[9E+09,9E+09,9E+09,9E+09,9E+09,9E+09]];
    CONST robtarget T201:=[[55.750402,39.462091,2.249551],[1.000000,0.000000,0.000000,0.000000],[0,0,-1,0],[9E+09,9E+09,9E+09,9E+09,9E+09,9E+09]];
    CONST robtarget T202:=[[57.250408,39.440997,2.249551],[1.000000,0.000000,0.000000,0.000000],[0,0,-1,0],[9E+09,9E+09,9E+09,9E+09,9E+09,9E+09]];
    CONST robtarget T203:=[[57.250408,71.973400,2.249551],[1.000000,0.000000,0.000000,0.000000],[0,0,-1,0],[9E+09,9E+09,9E+09,9E+09,9E+09,9E+09]];
    CONST robtarget T204:=[[58.750414,71.906869,2.249551],[1.000000,0.000000,0.000000,0.000000],[0,0,-1,0],[9E+09,9E+09,9E+09,9E+09,9E+09,9E+09]];
    CONST robtarget T205:=[[58.750414,39.536995,2.249551],[1.000000,0.000000,0.000000,0.000000],[0,0,-1,0],[9E+09,9E+09,9E+09,9E+09,9E+09,9E+09]];
    CONST robtarget T206:=[[60.250420,39.761602,2.249551],[1.000000,0.000000,0.000000,0.000000],[0,0,-1,0],[9E+09,9E+09,9E+09,9E+09,9E+09,9E+09]];
    CONST robtarget T207:=[[60.250420,71.805415,2.249551],[1.000000,0.000000,0.000000,0.000000],[0,0,-1,0],[9E+09,9E+09,9E+09,9E+09,9E+09,9E+09]];
    CONST robtarget T208:=[[61.750426,71.628887,2.249551],[1.000000,0.000000,0.000000,0.000000],[0,0,-1,0],[9E+09,9E+09,9E+09,9E+09,9E+09,9E+09]];
    CONST robtarget T209:=[[61.750426,40.150081,2.249551],[1.000000,0.000000,0.000000,0.000000],[0,0,-1,0],[9E+09,9E+09,9E+09,9E+09,9E+09,9E+09]];
    CONST robtarget T210:=[[63.250432,40.618904,2.249551],[1.000000,0.000000,0.000000,0.000000],[0,0,-1,0],[9E+09,9E+09,9E+09,9E+09,9E+09,9E+09]];
    CONST robtarget T211:=[[63.250432,71.246858,2.249551],[1.000000,0.000000,0.000000,0.000000],[0,0,-1,0],[9E+09,9E+09,9E+09,9E+09,9E+09,9E+09]];
    CONST robtarget T212:=[[64.750438,70.830826,2.249551],[1.000000,0.000000,0.000000,0.000000],[0,0,-1,0],[9E+09,9E+09,9E+09,9E+09,9E+09,9E+09]];
    CONST robtarget T213:=[[64.750438,41.202695,2.249551],[1.000000,0.000000,0.000000,0.000000],[0,0,-1,0],[9E+09,9E+09,9E+09,9E+09,9E+09,9E+09]];
    CONST robtarget T214:=[[66.250444,41.846848,2.249551],[1.000000,0.000000,0.000000,0.000000],[0,0,-1,0],[9E+09,9E+09,9E+09,9E+09,9E+09,9E+09]];
    CONST robtarget T215:=[[66.250444,70.007925,2.249551],[1.000000,0.000000,0.000000,0.000000],[0,0,-1,0],[9E+09,9E+09,9E+09,9E+09,9E+09,9E+09]];
    CONST robtarget T216:=[[67.750450,69.121513,2.249551],[1.000000,0.000000,0.000000,0.000000],[0,0,-1,0],[9E+09,9E+09,9E+09,9E+09,9E+09,9E+09]];
    CONST robtarget T217:=[[67.750450,42.607272,2.249551],[1.000000,0.000000,0.000000,0.000000],[0,0,-1,0],[9E+09,9E+09,9E+09,9E+09,9E+09,9E+09]];
    CONST robtarget T218:=[[69.250456,43.327801,2.249551],[1.000000,0.000000,0.000000,0.000000],[0,0,-1,0],[9E+09,9E+09,9E+09,9E+09,9E+09,9E+09]];
    CONST robtarget T219:=[[69.250456,67.989308,2.249551],[1.000000,0.000000,0.000000,0.000000],[0,0,-1,0],[9E+09,9E+09,9E+09,9E+09,9E+09,9E+09]];
    CONST robtarget T220:=[[70.750462,66.307133,2.249551],[1.000000,0.000000,0.000000,0.000000],[0,0,-1,0],[9E+09,9E+09,9E+09,9E+09,9E+09,9E+09]];
    CONST robtarget T221:=[[70.750462,44.569608,2.249551],[1.000000,0.000000,0.000000,0.000000],[0,0,-1,0],[9E+09,9E+09,9E+09,9E+09,9E+09,9E+09]];
    CONST robtarget T222:=[[72.250468,45.992999,2.249551],[1.000000,0.000000,0.000000,0.000000],[0,0,-1,0],[9E+09,9E+09,9E+09,9E+09,9E+09,9E+09]];
    CONST robtarget T223:=[[72.250468,64.081234,2.249551],[1.000000,0.000000,0.000000,0.000000],[0,0,-1,0],[9E+09,9E+09,9E+09,9E+09,9E+09,9E+09]];
    CONST robtarget T224:=[[73.750474,59.212343,2.249551],[1.000000,0.000000,0.000000,0.000000],[0,0,-1,0],[9E+09,9E+09,9E+09,9E+09,9E+09,9E+09]];
    CONST robtarget T225:=[[73.750474,48.399033,2.249551],[1.000000,0.000000,0.000000,0.000000],[0,0,-1,0],[9E+09,9E+09,9E+09,9E+09,9E+09,9E+09]];
    CONST robtarget T226:=[[74.500084,47.387823,2.749561],[1.000000,0.000000,0.000000,0.000000],[0,0,-1,0],[9E+09,9E+09,9E+09,9E+09,9E+09,9E+09]];
    CONST robtarget T227:=[[74.500084,58.421250,2.749561],[1.000000,0.000000,0.000000,0.000000],[0,0,-1,0],[9E+09,9E+09,9E+09,9E+09,9E+09,9E+09]];
    CONST robtarget T228:=[[74.500084,47.387823,2.749561],[1.000000,0.000000,0.000000,0.000000],[0,0,-1,0],[9E+09,9E+09,9E+09,9E+09,9E+09,9E+09]];
    CONST robtarget T229:=[[74.500084,58.421250,2.749561],[1.000000,0.000000,0.000000,0.000000],[0,0,-1,0],[9E+09,9E+09,9E+09,9E+09,9E+09,9E+09]];
    CONST robtarget T230:=[[73.000078,64.040830,2.749561],[1.000000,0.000000,0.000000,0.000000],[0,0,-1,0],[9E+09,9E+09,9E+09,9E+09,9E+09,9E+09]];
    CONST robtarget T231:=[[73.000078,45.431077,2.749561],[1.000000,0.000000,0.000000,0.000000],[0,0,-1,0],[9E+09,9E+09,9E+09,9E+09,9E+09,9E+09]];
    CONST robtarget T232:=[[71.500072,44.228710,2.749561],[1.000000,0.000000,0.000000,0.000000],[0,0,-1,0],[9E+09,9E+09,9E+09,9E+09,9E+09,9E+09]];
    CONST robtarget T233:=[[71.500072,66.412663,2.749561],[1.000000,0.000000,0.000000,0.000000],[0,0,-1,0],[9E+09,9E+09,9E+09,9E+09,9E+09,9E+09]];
    CONST robtarget T234:=[[70.000066,68.007397,2.749561],[1.000000,0.000000,0.000000,0.000000],[0,0,-1,0],[9E+09,9E+09,9E+09,9E+09,9E+09,9E+09]];
    CONST robtarget T235:=[[70.000066,43.032736,2.749561],[1.000000,0.000000,0.000000,0.000000],[0,0,-1,0],[9E+09,9E+09,9E+09,9E+09,9E+09,9E+09]];
    CONST robtarget T236:=[[68.500060,42.124213,2.749561],[1.000000,0.000000,0.000000,0.000000],[0,0,-1,0],[9E+09,9E+09,9E+09,9E+09,9E+09,9E+09]];
    CONST robtarget T237:=[[68.500060,69.277983,2.749561],[1.000000,0.000000,0.000000,0.000000],[0,0,-1,0],[9E+09,9E+09,9E+09,9E+09,9E+09,9E+09]];
    CONST robtarget T238:=[[67.000054,70.433873,2.749561],[1.000000,0.000000,0.000000,0.000000],[0,0,-1,0],[9E+09,9E+09,9E+09,9E+09,9E+09,9E+09]];
    CONST robtarget T239:=[[67.000054,41.370716,2.749561],[1.000000,0.000000,0.000000,0.000000],[0,0,-1,0],[9E+09,9E+09,9E+09,9E+09,9E+09,9E+09]];
    CONST robtarget T240:=[[65.500048,40.567590,2.749561],[1.000000,0.000000,0.000000,0.000000],[0,0,-1,0],[9E+09,9E+09,9E+09,9E+09,9E+09,9E+09]];
    CONST robtarget T241:=[[65.500048,71.261215,2.749561],[1.000000,0.000000,0.000000,0.000000],[0,0,-1,0],[9E+09,9E+09,9E+09,9E+09,9E+09,9E+09]];
    CONST robtarget T242:=[[64.000042,72.088557,2.749561],[1.000000,0.000000,0.000000,0.000000],[0,0,-1,0],[9E+09,9E+09,9E+09,9E+09,9E+09,9E+09]];
    CONST robtarget T243:=[[64.000042,39.975861,2.749561],[1.000000,0.000000,0.000000,0.000000],[0,0,-1,0],[9E+09,9E+09,9E+09,9E+09,9E+09,9E+09]];
    CONST robtarget T244:=[[62.500036,39.478997,2.749561],[1.000000,0.000000,0.000000,0.000000],[0,0,-1,0],[9E+09,9E+09,9E+09,9E+09,9E+09,9E+09]];
    CONST robtarget T245:=[[62.500036,72.394376,2.749561],[1.000000,0.000000,0.000000,0.000000],[0,0,-1,0],[9E+09,9E+09,9E+09,9E+09,9E+09,9E+09]];
    CONST robtarget T246:=[[61.000030,72.668403,2.749561],[1.000000,0.000000,0.000000,0.000000],[0,0,-1,0],[9E+09,9E+09,9E+09,9E+09,9E+09,9E+09]];
    CONST robtarget T247:=[[61.000030,39.158404,2.749561],[1.000000,0.000000,0.000000,0.000000],[0,0,-1,0],[9E+09,9E+09,9E+09,9E+09,9E+09,9E+09]];
    CONST robtarget T248:=[[59.500024,38.840635,2.749561],[1.000000,0.000000,0.000000,0.000000],[0,0,-1,0],[9E+09,9E+09,9E+09,9E+09,9E+09,9E+09]];
    CONST robtarget T249:=[[59.500024,72.748141,2.749561],[1.000000,0.000000,0.000000,0.000000],[0,0,-1,0],[9E+09,9E+09,9E+09,9E+09,9E+09,9E+09]];
    CONST robtarget T250:=[[58.000018,72.831262,2.749561],[1.000000,0.000000,0.000000,0.000000],[0,0,-1,0],[9E+09,9E+09,9E+09,9E+09,9E+09,9E+09]];
    CONST robtarget T251:=[[58.000018,38.730317,2.749561],[1.000000,0.000000,0.000000,0.000000],[0,0,-1,0],[9E+09,9E+09,9E+09,9E+09,9E+09,9E+09]];
    CONST robtarget T252:=[[56.500012,38.676982,2.749561],[1.000000,0.000000,0.000000,0.000000],[0,0,-1,0],[9E+09,9E+09,9E+09,9E+09,9E+09,9E+09]];
    CONST robtarget T253:=[[56.500012,72.883479,2.749561],[1.000000,0.000000,0.000000,0.000000],[0,0,-1,0],[9E+09,9E+09,9E+09,9E+09,9E+09,9E+09]];
    CONST robtarget T254:=[[55.000006,72.922065,2.749561],[1.000000,0.000000,0.000000,0.000000],[0,0,-1,0],[9E+09,9E+09,9E+09,9E+09,9E+09,9E+09]];
    CONST robtarget T255:=[[55.000006,38.677271,2.749561],[1.000000,0.000000,0.000000,0.000000],[0,0,-1,0],[9E+09,9E+09,9E+09,9E+09,9E+09,9E+09]];
    CONST robtarget T256:=[[53.500000,38.676982,2.749561],[1.000000,0.000000,0.000000,0.000000],[0,0,-1,0],[9E+09,9E+09,9E+09,9E+09,9E+09,9E+09]];
    CONST robtarget T257:=[[53.500000,72.883491,2.749561],[1.000000,0.000000,0.000000,0.000000],[0,0,-1,0],[9E+09,9E+09,9E+09,9E+09,9E+09,9E+09]];
    CONST robtarget T258:=[[51.999994,72.831262,2.749561],[1.000000,0.000000,0.000000,0.000000],[0,0,-1,0],[9E+09,9E+09,9E+09,9E+09,9E+09,9E+09]];
    CONST robtarget T259:=[[51.999994,38.730318,2.749561],[1.000000,0.000000,0.000000,0.000000],[0,0,-1,0],[9E+09,9E+09,9E+09,9E+09,9E+09,9E+09]];
    CONST robtarget T260:=[[50.499988,38.840635,2.749561],[1.000000,0.000000,0.000000,0.000000],[0,0,-1,0],[9E+09,9E+09,9E+09,9E+09,9E+09,9E+09]];
    CONST robtarget T261:=[[50.499988,72.748141,2.749561],[1.000000,0.000000,0.000000,0.000000],[0,0,-1,0],[9E+09,9E+09,9E+09,9E+09,9E+09,9E+09]];
    CONST robtarget T262:=[[48.999982,72.668403,2.749561],[1.000000,0.000000,0.000000,0.000000],[0,0,-1,0],[9E+09,9E+09,9E+09,9E+09,9E+09,9E+09]];
    CONST robtarget T263:=[[48.999982,39.158405,2.749561],[1.000000,0.000000,0.000000,0.000000],[0,0,-1,0],[9E+09,9E+09,9E+09,9E+09,9E+09,9E+09]];
    CONST robtarget T264:=[[47.499976,39.478997,2.749561],[1.000000,0.000000,0.000000,0.000000],[0,0,-1,0],[9E+09,9E+09,9E+09,9E+09,9E+09,9E+09]];
    CONST robtarget T265:=[[47.499976,72.394375,2.749561],[1.000000,0.000000,0.000000,0.000000],[0,0,-1,0],[9E+09,9E+09,9E+09,9E+09,9E+09,9E+09]];
    CONST robtarget T266:=[[45.999970,72.088555,2.749561],[1.000000,0.000000,0.000000,0.000000],[0,0,-1,0],[9E+09,9E+09,9E+09,9E+09,9E+09,9E+09]];
    CONST robtarget T267:=[[45.999970,39.975864,2.749561],[1.000000,0.000000,0.000000,0.000000],[0,0,-1,0],[9E+09,9E+09,9E+09,9E+09,9E+09,9E+09]];
    CONST robtarget T268:=[[44.499964,40.567596,2.749561],[1.000000,0.000000,0.000000,0.000000],[0,0,-1,0],[9E+09,9E+09,9E+09,9E+09,9E+09,9E+09]];
    CONST robtarget T269:=[[44.499964,71.261214,2.749561],[1.000000,0.000000,0.000000,0.000000],[0,0,-1,0],[9E+09,9E+09,9E+09,9E+09,9E+09,9E+09]];
    CONST robtarget T270:=[[42.999958,70.433872,2.749561],[1.000000,0.000000,0.000000,0.000000],[0,0,-1,0],[9E+09,9E+09,9E+09,9E+09,9E+09,9E+09]];
    CONST robtarget T271:=[[42.999958,41.370721,2.749561],[1.000000,0.000000,0.000000,0.000000],[0,0,-1,0],[9E+09,9E+09,9E+09,9E+09,9E+09,9E+09]];
    CONST robtarget T272:=[[41.499952,42.124214,2.749561],[1.000000,0.000000,0.000000,0.000000],[0,0,-1,0],[9E+09,9E+09,9E+09,9E+09,9E+09,9E+09]];
    CONST robtarget T273:=[[41.499952,69.277982,2.749561],[1.000000,0.000000,0.000000,0.000000],[0,0,-1,0],[9E+09,9E+09,9E+09,9E+09,9E+09,9E+09]];
    CONST robtarget T274:=[[39.999946,68.007395,2.749561],[1.000000,0.000000,0.000000,0.000000],[0,0,-1,0],[9E+09,9E+09,9E+09,9E+09,9E+09,9E+09]];
    CONST robtarget T275:=[[39.999946,43.032737,2.749561],[1.000000,0.000000,0.000000,0.000000],[0,0,-1,0],[9E+09,9E+09,9E+09,9E+09,9E+09,9E+09]];
    CONST robtarget T276:=[[38.499940,44.228713,2.749561],[1.000000,0.000000,0.000000,0.000000],[0,0,-1,0],[9E+09,9E+09,9E+09,9E+09,9E+09,9E+09]];
    CONST robtarget T277:=[[38.499940,66.413277,2.749561],[1.000000,0.000000,0.000000,0.000000],[0,0,-1,0],[9E+09,9E+09,9E+09,9E+09,9E+09,9E+09]];
    CONST robtarget T278:=[[36.999934,64.057909,2.749561],[1.000000,0.000000,0.000000,0.000000],[0,0,-1,0],[9E+09,9E+09,9E+09,9E+09,9E+09,9E+09]];
    CONST robtarget T279:=[[36.999934,45.431079,2.749561],[1.000000,0.000000,0.000000,0.000000],[0,0,-1,0],[9E+09,9E+09,9E+09,9E+09,9E+09,9E+09]];
    CONST robtarget T280:=[[35.499928,47.387823,2.749561],[1.000000,0.000000,0.000000,0.000000],[0,0,-1,0],[9E+09,9E+09,9E+09,9E+09,9E+09,9E+09]];
    CONST robtarget T281:=[[35.499928,58.459385,2.749561],[1.000000,0.000000,0.000000,0.000000],[0,0,-1,0],[9E+09,9E+09,9E+09,9E+09,9E+09,9E+09]];
    CONST robtarget T282:=[[34.749925,48.064691,3.249571],[1.000000,0.000000,0.000000,0.000000],[0,0,-1,0],[9E+09,9E+09,9E+09,9E+09,9E+09,9E+09]];
    CONST robtarget T283:=[[34.749925,56.866082,3.249571],[1.000000,0.000000,0.000000,0.000000],[0,0,-1,0],[9E+09,9E+09,9E+09,9E+09,9E+09,9E+09]];
    CONST robtarget T284:=[[34.749925,48.064691,3.249571],[1.000000,0.000000,0.000000,0.000000],[0,0,-1,0],[9E+09,9E+09,9E+09,9E+09,9E+09,9E+09]];
    CONST robtarget T285:=[[34.749925,56.866082,3.249571],[1.000000,0.000000,0.000000,0.000000],[0,0,-1,0],[9E+09,9E+09,9E+09,9E+09,9E+09,9E+09]];
    CONST robtarget T286:=[[36.249931,62.796554,3.249571],[1.000000,0.000000,0.000000,0.000000],[0,0,-1,0],[9E+09,9E+09,9E+09,9E+09,9E+09,9E+09]];
    CONST robtarget T287:=[[36.249931,45.294379,3.249571],[1.000000,0.000000,0.000000,0.000000],[0,0,-1,0],[9E+09,9E+09,9E+09,9E+09,9E+09,9E+09]];
    CONST robtarget T288:=[[37.749937,43.856197,3.249571],[1.000000,0.000000,0.000000,0.000000],[0,0,-1,0],[9E+09,9E+09,9E+09,9E+09,9E+09,9E+09]];
    CONST robtarget T289:=[[37.749937,66.109809,3.249571],[1.000000,0.000000,0.000000,0.000000],[0,0,-1,0],[9E+09,9E+09,9E+09,9E+09,9E+09,9E+09]];
    CONST robtarget T290:=[[39.249943,68.023443,3.249571],[1.000000,0.000000,0.000000,0.000000],[0,0,-1,0],[9E+09,9E+09,9E+09,9E+09,9E+09,9E+09]];
    CONST robtarget T291:=[[39.249943,42.775533,3.249571],[1.000000,0.000000,0.000000,0.000000],[0,0,-1,0],[9E+09,9E+09,9E+09,9E+09,9E+09,9E+09]];
    CONST robtarget T292:=[[40.749949,41.794433,3.249571],[1.000000,0.000000,0.000000,0.000000],[0,0,-1,0],[9E+09,9E+09,9E+09,9E+09,9E+09,9E+09]];
    CONST robtarget T293:=[[40.749949,69.250863,3.249571],[1.000000,0.000000,0.000000,0.000000],[0,0,-1,0],[9E+09,9E+09,9E+09,9E+09,9E+09,9E+09]];
    CONST robtarget T294:=[[42.249955,70.401290,3.249571],[1.000000,0.000000,0.000000,0.000000],[0,0,-1,0],[9E+09,9E+09,9E+09,9E+09,9E+09,9E+09]];
    CONST robtarget T295:=[[42.249955,40.894833,3.249571],[1.000000,0.000000,0.000000,0.000000],[0,0,-1,0],[9E+09,9E+09,9E+09,9E+09,9E+09,9E+09]];
    CONST robtarget T296:=[[43.749961,40.199626,3.249571],[1.000000,0.000000,0.000000,0.000000],[0,0,-1,0],[9E+09,9E+09,9E+09,9E+09,9E+09,9E+09]];
    CONST robtarget T297:=[[43.749961,71.522552,3.249571],[1.000000,0.000000,0.000000,0.000000],[0,0,-1,0],[9E+09,9E+09,9E+09,9E+09,9E+09,9E+09]];
    CONST robtarget T298:=[[45.249967,72.265960,3.249571],[1.000000,0.000000,0.000000,0.000000],[0,0,-1,0],[9E+09,9E+09,9E+09,9E+09,9E+09,9E+09]];
    CONST robtarget T299:=[[45.249967,39.594760,3.249571],[1.000000,0.000000,0.000000,0.000000],[0,0,-1,0],[9E+09,9E+09,9E+09,9E+09,9E+09,9E+09]];
    CONST robtarget T300:=[[46.749973,39.094363,3.249571],[1.000000,0.000000,0.000000,0.000000],[0,0,-1,0],[9E+09,9E+09,9E+09,9E+09,9E+09,9E+09]];
    CONST robtarget T301:=[[46.749973,72.924257,3.249571],[1.000000,0.000000,0.000000,0.000000],[0,0,-1,0],[9E+09,9E+09,9E+09,9E+09,9E+09,9E+09]];
    CONST robtarget T302:=[[48.249979,73.216923,3.249571],[1.000000,0.000000,0.000000,0.000000],[0,0,-1,0],[9E+09,9E+09,9E+09,9E+09,9E+09,9E+09]];
    CONST robtarget T303:=[[48.249979,38.736257,3.249571],[1.000000,0.000000,0.000000,0.000000],[0,0,-1,0],[9E+09,9E+09,9E+09,9E+09,9E+09,9E+09]];
    CONST robtarget T304:=[[49.749985,38.418924,3.249571],[1.000000,0.000000,0.000000,0.000000],[0,0,-1,0],[9E+09,9E+09,9E+09,9E+09,9E+09,9E+09]];
    CONST robtarget T305:=[[49.749985,73.423277,3.249571],[1.000000,0.000000,0.000000,0.000000],[0,0,-1,0],[9E+09,9E+09,9E+09,9E+09,9E+09,9E+09]];
    CONST robtarget T306:=[[51.249991,73.504461,3.249571],[1.000000,0.000000,0.000000,0.000000],[0,0,-1,0],[9E+09,9E+09,9E+09,9E+09,9E+09,9E+09]];
    CONST robtarget T307:=[[51.249991,38.215233,3.249571],[1.000000,0.000000,0.000000,0.000000],[0,0,-1,0],[9E+09,9E+09,9E+09,9E+09,9E+09,9E+09]];
    CONST robtarget T308:=[[52.749997,38.122806,3.249571],[1.000000,0.000000,0.000000,0.000000],[0,0,-1,0],[9E+09,9E+09,9E+09,9E+09,9E+09,9E+09]];
    CONST robtarget T309:=[[52.749997,73.592243,3.249571],[1.000000,0.000000,0.000000,0.000000],[0,0,-1,0],[9E+09,9E+09,9E+09,9E+09,9E+09,9E+09]];
    CONST robtarget T310:=[[54.250003,73.642177,3.249571],[1.000000,0.000000,0.000000,0.000000],[0,0,-1,0],[9E+09,9E+09,9E+09,9E+09,9E+09,9E+09]];
    CONST robtarget T311:=[[54.250003,38.121437,3.249571],[1.000000,0.000000,0.000000,0.000000],[0,0,-1,0],[9E+09,9E+09,9E+09,9E+09,9E+09,9E+09]];
    CONST robtarget T312:=[[55.750009,38.121437,3.249571],[1.000000,0.000000,0.000000,0.000000],[0,0,-1,0],[9E+09,9E+09,9E+09,9E+09,9E+09,9E+09]];
    CONST robtarget T313:=[[55.750009,73.642177,3.249571],[1.000000,0.000000,0.000000,0.000000],[0,0,-1,0],[9E+09,9E+09,9E+09,9E+09,9E+09,9E+09]];
    CONST robtarget T314:=[[57.250015,73.592243,3.249571],[1.000000,0.000000,0.000000,0.000000],[0,0,-1,0],[9E+09,9E+09,9E+09,9E+09,9E+09,9E+09]];
    CONST robtarget T315:=[[57.250015,38.122806,3.249571],[1.000000,0.000000,0.000000,0.000000],[0,0,-1,0],[9E+09,9E+09,9E+09,9E+09,9E+09,9E+09]];
    CONST robtarget T316:=[[58.750021,38.215233,3.249571],[1.000000,0.000000,0.000000,0.000000],[0,0,-1,0],[9E+09,9E+09,9E+09,9E+09,9E+09,9E+09]];
    CONST robtarget T317:=[[58.750021,73.504461,3.249571],[1.000000,0.000000,0.000000,0.000000],[0,0,-1,0],[9E+09,9E+09,9E+09,9E+09,9E+09,9E+09]];
    CONST robtarget T318:=[[60.250027,73.423277,3.249571],[1.000000,0.000000,0.000000,0.000000],[0,0,-1,0],[9E+09,9E+09,9E+09,9E+09,9E+09,9E+09]];
    CONST robtarget T319:=[[60.250027,38.418924,3.249571],[1.000000,0.000000,0.000000,0.000000],[0,0,-1,0],[9E+09,9E+09,9E+09,9E+09,9E+09,9E+09]];
    CONST robtarget T320:=[[61.750033,38.736257,3.249571],[1.000000,0.000000,0.000000,0.000000],[0,0,-1,0],[9E+09,9E+09,9E+09,9E+09,9E+09,9E+09]];
    CONST robtarget T321:=[[61.750033,73.216924,3.249571],[1.000000,0.000000,0.000000,0.000000],[0,0,-1,0],[9E+09,9E+09,9E+09,9E+09,9E+09,9E+09]];
    CONST robtarget T322:=[[63.250039,72.924257,3.249571],[1.000000,0.000000,0.000000,0.000000],[0,0,-1,0],[9E+09,9E+09,9E+09,9E+09,9E+09,9E+09]];
    CONST robtarget T323:=[[63.250039,39.094363,3.249571],[1.000000,0.000000,0.000000,0.000000],[0,0,-1,0],[9E+09,9E+09,9E+09,9E+09,9E+09,9E+09]];
    CONST robtarget T324:=[[64.750045,39.594757,3.249571],[1.000000,0.000000,0.000000,0.000000],[0,0,-1,0],[9E+09,9E+09,9E+09,9E+09,9E+09,9E+09]];
    CONST robtarget T325:=[[64.750045,72.265963,3.249571],[1.000000,0.000000,0.000000,0.000000],[0,0,-1,0],[9E+09,9E+09,9E+09,9E+09,9E+09,9E+09]];
    CONST robtarget T326:=[[66.250051,71.522553,3.249571],[1.000000,0.000000,0.000000,0.000000],[0,0,-1,0],[9E+09,9E+09,9E+09,9E+09,9E+09,9E+09]];
    CONST robtarget T327:=[[66.250051,40.199621,3.249571],[1.000000,0.000000,0.000000,0.000000],[0,0,-1,0],[9E+09,9E+09,9E+09,9E+09,9E+09,9E+09]];
    CONST robtarget T328:=[[67.750057,40.894831,3.249571],[1.000000,0.000000,0.000000,0.000000],[0,0,-1,0],[9E+09,9E+09,9E+09,9E+09,9E+09,9E+09]];
    CONST robtarget T329:=[[67.750057,70.401291,3.249571],[1.000000,0.000000,0.000000,0.000000],[0,0,-1,0],[9E+09,9E+09,9E+09,9E+09,9E+09,9E+09]];
    CONST robtarget T330:=[[69.250063,69.250864,3.249571],[1.000000,0.000000,0.000000,0.000000],[0,0,-1,0],[9E+09,9E+09,9E+09,9E+09,9E+09,9E+09]];
    CONST robtarget T331:=[[69.250063,41.794432,3.249571],[1.000000,0.000000,0.000000,0.000000],[0,0,-1,0],[9E+09,9E+09,9E+09,9E+09,9E+09,9E+09]];
    CONST robtarget T332:=[[70.750069,42.775532,3.249571],[1.000000,0.000000,0.000000,0.000000],[0,0,-1,0],[9E+09,9E+09,9E+09,9E+09,9E+09,9E+09]];
    CONST robtarget T333:=[[70.750069,68.023444,3.249571],[1.000000,0.000000,0.000000,0.000000],[0,0,-1,0],[9E+09,9E+09,9E+09,9E+09,9E+09,9E+09]];
    CONST robtarget T334:=[[72.250075,66.107177,3.249571],[1.000000,0.000000,0.000000,0.000000],[0,0,-1,0],[9E+09,9E+09,9E+09,9E+09,9E+09,9E+09]];
    CONST robtarget T335:=[[72.250075,43.856194,3.249571],[1.000000,0.000000,0.000000,0.000000],[0,0,-1,0],[9E+09,9E+09,9E+09,9E+09,9E+09,9E+09]];
    CONST robtarget T336:=[[73.750081,45.294376,3.249571],[1.000000,0.000000,0.000000,0.000000],[0,0,-1,0],[9E+09,9E+09,9E+09,9E+09,9E+09,9E+09]];
    CONST robtarget T337:=[[73.750081,62.771061,3.249571],[1.000000,0.000000,0.000000,0.000000],[0,0,-1,0],[9E+09,9E+09,9E+09,9E+09,9E+09,9E+09]];
    CONST robtarget T338:=[[75.250087,56.839386,3.249571],[1.000000,0.000000,0.000000,0.000000],[0,0,-1,0],[9E+09,9E+09,9E+09,9E+09,9E+09,9E+09]];
    CONST robtarget T339:=[[75.250087,48.064693,3.249571],[1.000000,0.000000,0.000000,0.000000],[0,0,-1,0],[9E+09,9E+09,9E+09,9E+09,9E+09,9E+09]];
    CONST robtarget T340:=[[75.250088,46.769603,3.749581],[1.000000,0.000000,0.000000,0.000000],[0,0,-1,0],[9E+09,9E+09,9E+09,9E+09,9E+09,9E+09]];
    CONST robtarget T341:=[[75.250088,58.240395,3.749581],[1.000000,0.000000,0.000000,0.000000],[0,0,-1,0],[9E+09,9E+09,9E+09,9E+09,9E+09,9E+09]];
    CONST robtarget T342:=[[75.250088,46.769603,3.749581],[1.000000,0.000000,0.000000,0.000000],[0,0,-1,0],[9E+09,9E+09,9E+09,9E+09,9E+09,9E+09]];
    CONST robtarget T343:=[[75.250088,58.240395,3.749581],[1.000000,0.000000,0.000000,0.000000],[0,0,-1,0],[9E+09,9E+09,9E+09,9E+09,9E+09,9E+09]];
    CONST robtarget T344:=[[73.750082,63.420809,3.749581],[1.000000,0.000000,0.000000,0.000000],[0,0,-1,0],[9E+09,9E+09,9E+09,9E+09,9E+09,9E+09]];
    CONST robtarget T345:=[[73.750082,44.665271,3.749581],[1.000000,0.000000,0.000000,0.000000],[0,0,-1,0],[9E+09,9E+09,9E+09,9E+09,9E+09,9E+09]];
    CONST robtarget T346:=[[72.250076,43.193451,3.749581],[1.000000,0.000000,0.000000,0.000000],[0,0,-1,0],[9E+09,9E+09,9E+09,9E+09,9E+09,9E+09]];
    CONST robtarget T347:=[[72.250076,66.449967,3.749581],[1.000000,0.000000,0.000000,0.000000],[0,0,-1,0],[9E+09,9E+09,9E+09,9E+09,9E+09,9E+09]];
    CONST robtarget T348:=[[70.750070,68.419833,3.749581],[1.000000,0.000000,0.000000,0.000000],[0,0,-1,0],[9E+09,9E+09,9E+09,9E+09,9E+09,9E+09]];
    CONST robtarget T349:=[[70.750070,42.087470,3.749581],[1.000000,0.000000,0.000000,0.000000],[0,0,-1,0],[9E+09,9E+09,9E+09,9E+09,9E+09,9E+09]];
    CONST robtarget T350:=[[69.250064,41.130024,3.749581],[1.000000,0.000000,0.000000,0.000000],[0,0,-1,0],[9E+09,9E+09,9E+09,9E+09,9E+09,9E+09]];
    CONST robtarget T351:=[[69.250064,69.830682,3.749581],[1.000000,0.000000,0.000000,0.000000],[0,0,-1,0],[9E+09,9E+09,9E+09,9E+09,9E+09,9E+09]];
    CONST robtarget T352:=[[67.750058,70.887914,3.749581],[1.000000,0.000000,0.000000,0.000000],[0,0,-1,0],[9E+09,9E+09,9E+09,9E+09,9E+09,9E+09]];
    CONST robtarget T353:=[[67.750058,40.269507,3.749581],[1.000000,0.000000,0.000000,0.000000],[0,0,-1,0],[9E+09,9E+09,9E+09,9E+09,9E+09,9E+09]];
    CONST robtarget T354:=[[66.250052,39.569745,3.749581],[1.000000,0.000000,0.000000,0.000000],[0,0,-1,0],[9E+09,9E+09,9E+09,9E+09,9E+09,9E+09]];
    CONST robtarget T355:=[[66.250052,72.006828,3.749581],[1.000000,0.000000,0.000000,0.000000],[0,0,-1,0],[9E+09,9E+09,9E+09,9E+09,9E+09,9E+09]];
    CONST robtarget T356:=[[64.750046,72.779280,3.749581],[1.000000,0.000000,0.000000,0.000000],[0,0,-1,0],[9E+09,9E+09,9E+09,9E+09,9E+09,9E+09]];
    CONST robtarget T357:=[[64.750046,38.962751,3.749581],[1.000000,0.000000,0.000000,0.000000],[0,0,-1,0],[9E+09,9E+09,9E+09,9E+09,9E+09,9E+09]];
    CONST robtarget T358:=[[63.250040,38.481957,3.749581],[1.000000,0.000000,0.000000,0.000000],[0,0,-1,0],[9E+09,9E+09,9E+09,9E+09,9E+09,9E+09]];
    CONST robtarget T359:=[[63.250040,73.580420,3.749581],[1.000000,0.000000,0.000000,0.000000],[0,0,-1,0],[9E+09,9E+09,9E+09,9E+09,9E+09,9E+09]];
    CONST robtarget T360:=[[61.750034,73.879904,3.749581],[1.000000,0.000000,0.000000,0.000000],[0,0,-1,0],[9E+09,9E+09,9E+09,9E+09,9E+09,9E+09]];
    CONST robtarget T361:=[[61.750034,38.126080,3.749581],[1.000000,0.000000,0.000000,0.000000],[0,0,-1,0],[9E+09,9E+09,9E+09,9E+09,9E+09,9E+09]];
    CONST robtarget T362:=[[60.250028,37.843736,3.749581],[1.000000,0.000000,0.000000,0.000000],[0,0,-1,0],[9E+09,9E+09,9E+09,9E+09,9E+09,9E+09]];
    CONST robtarget T363:=[[60.250028,74.116070,3.749581],[1.000000,0.000000,0.000000,0.000000],[0,0,-1,0],[9E+09,9E+09,9E+09,9E+09,9E+09,9E+09]];
    CONST robtarget T364:=[[58.750022,74.193872,3.749581],[1.000000,0.000000,0.000000,0.000000],[0,0,-1,0],[9E+09,9E+09,9E+09,9E+09,9E+09,9E+09]];
    CONST robtarget T365:=[[58.750022,37.644990,3.749581],[1.000000,0.000000,0.000000,0.000000],[0,0,-1,0],[9E+09,9E+09,9E+09,9E+09,9E+09,9E+09]];
    CONST robtarget T366:=[[57.250016,37.565151,3.749581],[1.000000,0.000000,0.000000,0.000000],[0,0,-1,0],[9E+09,9E+09,9E+09,9E+09,9E+09,9E+09]];
    CONST robtarget T367:=[[57.250016,74.275310,3.749581],[1.000000,0.000000,0.000000,0.000000],[0,0,-1,0],[9E+09,9E+09,9E+09,9E+09,9E+09,9E+09]];
    CONST robtarget T368:=[[55.750010,74.353482,3.749581],[1.000000,0.000000,0.000000,0.000000],[0,0,-1,0],[9E+09,9E+09,9E+09,9E+09,9E+09,9E+09]];
    CONST robtarget T369:=[[55.750010,37.565747,3.749581],[1.000000,0.000000,0.000000,0.000000],[0,0,-1,0],[9E+09,9E+09,9E+09,9E+09,9E+09,9E+09]];
    CONST robtarget T370:=[[54.250004,37.565747,3.749581],[1.000000,0.000000,0.000000,0.000000],[0,0,-1,0],[9E+09,9E+09,9E+09,9E+09,9E+09,9E+09]];
    CONST robtarget T371:=[[54.250004,74.353482,3.749581],[1.000000,0.000000,0.000000,0.000000],[0,0,-1,0],[9E+09,9E+09,9E+09,9E+09,9E+09,9E+09]];
    CONST robtarget T372:=[[52.749998,74.275310,3.749581],[1.000000,0.000000,0.000000,0.000000],[0,0,-1,0],[9E+09,9E+09,9E+09,9E+09,9E+09,9E+09]];
    CONST robtarget T373:=[[52.749998,37.565151,3.749581],[1.000000,0.000000,0.000000,0.000000],[0,0,-1,0],[9E+09,9E+09,9E+09,9E+09,9E+09,9E+09]];
    CONST robtarget T374:=[[51.249992,37.644990,3.749581],[1.000000,0.000000,0.000000,0.000000],[0,0,-1,0],[9E+09,9E+09,9E+09,9E+09,9E+09,9E+09]];
    CONST robtarget T375:=[[51.249992,74.193872,3.749581],[1.000000,0.000000,0.000000,0.000000],[0,0,-1,0],[9E+09,9E+09,9E+09,9E+09,9E+09,9E+09]];
    CONST robtarget T376:=[[49.749986,74.116070,3.749581],[1.000000,0.000000,0.000000,0.000000],[0,0,-1,0],[9E+09,9E+09,9E+09,9E+09,9E+09,9E+09]];
    CONST robtarget T377:=[[49.749986,37.843736,3.749581],[1.000000,0.000000,0.000000,0.000000],[0,0,-1,0],[9E+09,9E+09,9E+09,9E+09,9E+09,9E+09]];
    CONST robtarget T378:=[[48.249980,38.126081,3.749581],[1.000000,0.000000,0.000000,0.000000],[0,0,-1,0],[9E+09,9E+09,9E+09,9E+09,9E+09,9E+09]];
    CONST robtarget T379:=[[48.249980,73.879904,3.749581],[1.000000,0.000000,0.000000,0.000000],[0,0,-1,0],[9E+09,9E+09,9E+09,9E+09,9E+09,9E+09]];
    CONST robtarget T380:=[[46.749974,73.580420,3.749581],[1.000000,0.000000,0.000000,0.000000],[0,0,-1,0],[9E+09,9E+09,9E+09,9E+09,9E+09,9E+09]];
    CONST robtarget T381:=[[46.749974,38.481957,3.749581],[1.000000,0.000000,0.000000,0.000000],[0,0,-1,0],[9E+09,9E+09,9E+09,9E+09,9E+09,9E+09]];
    CONST robtarget T382:=[[45.249968,38.962753,3.749581],[1.000000,0.000000,0.000000,0.000000],[0,0,-1,0],[9E+09,9E+09,9E+09,9E+09,9E+09,9E+09]];
    CONST robtarget T383:=[[45.249968,72.779274,3.749581],[1.000000,0.000000,0.000000,0.000000],[0,0,-1,0],[9E+09,9E+09,9E+09,9E+09,9E+09,9E+09]];
    CONST robtarget T384:=[[43.749962,72.006826,3.749581],[1.000000,0.000000,0.000000,0.000000],[0,0,-1,0],[9E+09,9E+09,9E+09,9E+09,9E+09,9E+09]];
    CONST robtarget T385:=[[43.749962,39.569747,3.749581],[1.000000,0.000000,0.000000,0.000000],[0,0,-1,0],[9E+09,9E+09,9E+09,9E+09,9E+09,9E+09]];
    CONST robtarget T386:=[[42.249956,40.269508,3.749581],[1.000000,0.000000,0.000000,0.000000],[0,0,-1,0],[9E+09,9E+09,9E+09,9E+09,9E+09,9E+09]];
    CONST robtarget T387:=[[42.249956,70.887914,3.749581],[1.000000,0.000000,0.000000,0.000000],[0,0,-1,0],[9E+09,9E+09,9E+09,9E+09,9E+09,9E+09]];
    CONST robtarget T388:=[[40.749950,69.830682,3.749581],[1.000000,0.000000,0.000000,0.000000],[0,0,-1,0],[9E+09,9E+09,9E+09,9E+09,9E+09,9E+09]];
    CONST robtarget T389:=[[40.749950,41.130024,3.749581],[1.000000,0.000000,0.000000,0.000000],[0,0,-1,0],[9E+09,9E+09,9E+09,9E+09,9E+09,9E+09]];
    CONST robtarget T390:=[[39.249944,42.087470,3.749581],[1.000000,0.000000,0.000000,0.000000],[0,0,-1,0],[9E+09,9E+09,9E+09,9E+09,9E+09,9E+09]];
    CONST robtarget T391:=[[39.249944,68.419833,3.749581],[1.000000,0.000000,0.000000,0.000000],[0,0,-1,0],[9E+09,9E+09,9E+09,9E+09,9E+09,9E+09]];
    CONST robtarget T392:=[[37.749938,66.451990,3.749581],[1.000000,0.000000,0.000000,0.000000],[0,0,-1,0],[9E+09,9E+09,9E+09,9E+09,9E+09,9E+09]];
    CONST robtarget T393:=[[37.749938,43.193453,3.749581],[1.000000,0.000000,0.000000,0.000000],[0,0,-1,0],[9E+09,9E+09,9E+09,9E+09,9E+09,9E+09]];
    CONST robtarget T394:=[[36.249932,44.665272,3.749581],[1.000000,0.000000,0.000000,0.000000],[0,0,-1,0],[9E+09,9E+09,9E+09,9E+09,9E+09,9E+09]];
    CONST robtarget T395:=[[36.249932,63.436566,3.749581],[1.000000,0.000000,0.000000,0.000000],[0,0,-1,0],[9E+09,9E+09,9E+09,9E+09,9E+09,9E+09]];
    CONST robtarget T396:=[[34.749926,58.263819,3.749581],[1.000000,0.000000,0.000000,0.000000],[0,0,-1,0],[9E+09,9E+09,9E+09,9E+09,9E+09,9E+09]];
    CONST robtarget T397:=[[34.749926,46.769601,3.749581],[1.000000,0.000000,0.000000,0.000000],[0,0,-1,0],[9E+09,9E+09,9E+09,9E+09,9E+09,9E+09]];
    CONST robtarget T398:=[[33.999923,47.259734,4.249591],[1.000000,0.000000,0.000000,0.000000],[0,0,-1,0],[9E+09,9E+09,9E+09,9E+09,9E+09,9E+09]];
    CONST robtarget T399:=[[33.999923,56.747668,4.249591],[1.000000,0.000000,0.000000,0.000000],[0,0,-1,0],[9E+09,9E+09,9E+09,9E+09,9E+09,9E+09]];
    CONST robtarget T400:=[[33.999923,47.259734,4.249591],[1.000000,0.000000,0.000000,0.000000],[0,0,-1,0],[9E+09,9E+09,9E+09,9E+09,9E+09,9E+09]];
    CONST robtarget T401:=[[33.999923,56.747668,4.249591],[1.000000,0.000000,0.000000,0.000000],[0,0,-1,0],[9E+09,9E+09,9E+09,9E+09,9E+09,9E+09]];
    CONST robtarget T402:=[[35.499929,62.144514,4.249591],[1.000000,0.000000,0.000000,0.000000],[0,0,-1,0],[9E+09,9E+09,9E+09,9E+09,9E+09,9E+09]];
    CONST robtarget T403:=[[35.499929,44.766401,4.249591],[1.000000,0.000000,0.000000,0.000000],[0,0,-1,0],[9E+09,9E+09,9E+09,9E+09,9E+09,9E+09]];
    CONST robtarget T404:=[[36.999935,43.288408,4.249591],[1.000000,0.000000,0.000000,0.000000],[0,0,-1,0],[9E+09,9E+09,9E+09,9E+09,9E+09,9E+09]];
    CONST robtarget T405:=[[36.999935,65.778009,4.249591],[1.000000,0.000000,0.000000,0.000000],[0,0,-1,0],[9E+09,9E+09,9E+09,9E+09,9E+09,9E+09]];
    CONST robtarget T406:=[[38.499941,67.838098,4.249591],[1.000000,0.000000,0.000000,0.000000],[0,0,-1,0],[9E+09,9E+09,9E+09,9E+09,9E+09,9E+09]];
    CONST robtarget T407:=[[38.499941,42.013796,4.249591],[1.000000,0.000000,0.000000,0.000000],[0,0,-1,0],[9E+09,9E+09,9E+09,9E+09,9E+09,9E+09]];
    CONST robtarget T408:=[[39.999947,40.997439,4.249591],[1.000000,0.000000,0.000000,0.000000],[0,0,-1,0],[9E+09,9E+09,9E+09,9E+09,9E+09,9E+09]];
    CONST robtarget T409:=[[39.999947,69.500161,4.249591],[1.000000,0.000000,0.000000,0.000000],[0,0,-1,0],[9E+09,9E+09,9E+09,9E+09,9E+09,9E+09]];
    CONST robtarget T410:=[[41.499953,70.844693,4.249591],[1.000000,0.000000,0.000000,0.000000],[0,0,-1,0],[9E+09,9E+09,9E+09,9E+09,9E+09,9E+09]];
    CONST robtarget T411:=[[41.499953,40.066520,4.249591],[1.000000,0.000000,0.000000,0.000000],[0,0,-1,0],[9E+09,9E+09,9E+09,9E+09,9E+09,9E+09]];
    CONST robtarget T412:=[[42.999959,39.295226,4.249591],[1.000000,0.000000,0.000000,0.000000],[0,0,-1,0],[9E+09,9E+09,9E+09,9E+09,9E+09,9E+09]];
    CONST robtarget T413:=[[42.999959,71.924941,4.249591],[1.000000,0.000000,0.000000,0.000000],[0,0,-1,0],[9E+09,9E+09,9E+09,9E+09,9E+09,9E+09]];
    CONST robtarget T414:=[[44.499965,72.939569,4.249591],[1.000000,0.000000,0.000000,0.000000],[0,0,-1,0],[9E+09,9E+09,9E+09,9E+09,9E+09,9E+09]];
    CONST robtarget T415:=[[44.499965,38.592265,4.249591],[1.000000,0.000000,0.000000,0.000000],[0,0,-1,0],[9E+09,9E+09,9E+09,9E+09,9E+09,9E+09]];
    CONST robtarget T416:=[[45.999971,38.097323,4.249591],[1.000000,0.000000,0.000000,0.000000],[0,0,-1,0],[9E+09,9E+09,9E+09,9E+09,9E+09,9E+09]];
    CONST robtarget T417:=[[45.999971,73.715025,4.249591],[1.000000,0.000000,0.000000,0.000000],[0,0,-1,0],[9E+09,9E+09,9E+09,9E+09,9E+09,9E+09]];
    CONST robtarget T418:=[[47.499977,74.230219,4.249591],[1.000000,0.000000,0.000000,0.000000],[0,0,-1,0],[9E+09,9E+09,9E+09,9E+09,9E+09,9E+09]];
    CONST robtarget T419:=[[47.499977,37.641989,4.249591],[1.000000,0.000000,0.000000,0.000000],[0,0,-1,0],[9E+09,9E+09,9E+09,9E+09,9E+09,9E+09]];
    CONST robtarget T420:=[[48.999983,37.389818,4.249591],[1.000000,0.000000,0.000000,0.000000],[0,0,-1,0],[9E+09,9E+09,9E+09,9E+09,9E+09,9E+09]];
    CONST robtarget T421:=[[48.999983,74.473107,4.249591],[1.000000,0.000000,0.000000,0.000000],[0,0,-1,0],[9E+09,9E+09,9E+09,9E+09,9E+09,9E+09]];
    CONST robtarget T422:=[[50.499989,74.636276,4.249591],[1.000000,0.000000,0.000000,0.000000],[0,0,-1,0],[9E+09,9E+09,9E+09,9E+09,9E+09,9E+09]];
    CONST robtarget T423:=[[50.499989,37.129906,4.249591],[1.000000,0.000000,0.000000,0.000000],[0,0,-1,0],[9E+09,9E+09,9E+09,9E+09,9E+09,9E+09]];
    CONST robtarget T424:=[[51.999995,37.046902,4.249591],[1.000000,0.000000,0.000000,0.000000],[0,0,-1,0],[9E+09,9E+09,9E+09,9E+09,9E+09,9E+09]];
    CONST robtarget T425:=[[51.999995,74.714103,4.249591],[1.000000,0.000000,0.000000,0.000000],[0,0,-1,0],[9E+09,9E+09,9E+09,9E+09,9E+09,9E+09]];
    CONST robtarget T426:=[[53.500001,74.811282,4.249591],[1.000000,0.000000,0.000000,0.000000],[0,0,-1,0],[9E+09,9E+09,9E+09,9E+09,9E+09,9E+09]];
    CONST robtarget T427:=[[53.500001,37.008909,4.249591],[1.000000,0.000000,0.000000,0.000000],[0,0,-1,0],[9E+09,9E+09,9E+09,9E+09,9E+09,9E+09]];
    CONST robtarget T428:=[[55.000007,37.010202,4.249591],[1.000000,0.000000,0.000000,0.000000],[0,0,-1,0],[9E+09,9E+09,9E+09,9E+09,9E+09,9E+09]];
    CONST robtarget T429:=[[55.000007,74.887695,4.249591],[1.000000,0.000000,0.000000,0.000000],[0,0,-1,0],[9E+09,9E+09,9E+09,9E+09,9E+09,9E+09]];
    CONST robtarget T430:=[[56.500013,74.811282,4.249591],[1.000000,0.000000,0.000000,0.000000],[0,0,-1,0],[9E+09,9E+09,9E+09,9E+09,9E+09,9E+09]];
    CONST robtarget T431:=[[56.500013,37.008909,4.249591],[1.000000,0.000000,0.000000,0.000000],[0,0,-1,0],[9E+09,9E+09,9E+09,9E+09,9E+09,9E+09]];
    CONST robtarget T432:=[[58.000019,37.046902,4.249591],[1.000000,0.000000,0.000000,0.000000],[0,0,-1,0],[9E+09,9E+09,9E+09,9E+09,9E+09,9E+09]];
    CONST robtarget T433:=[[58.000019,74.714103,4.249591],[1.000000,0.000000,0.000000,0.000000],[0,0,-1,0],[9E+09,9E+09,9E+09,9E+09,9E+09,9E+09]];
    CONST robtarget T434:=[[59.500025,74.636276,4.249591],[1.000000,0.000000,0.000000,0.000000],[0,0,-1,0],[9E+09,9E+09,9E+09,9E+09,9E+09,9E+09]];
    CONST robtarget T435:=[[59.500025,37.129906,4.249591],[1.000000,0.000000,0.000000,0.000000],[0,0,-1,0],[9E+09,9E+09,9E+09,9E+09,9E+09,9E+09]];
    CONST robtarget T436:=[[61.000031,37.389818,4.249591],[1.000000,0.000000,0.000000,0.000000],[0,0,-1,0],[9E+09,9E+09,9E+09,9E+09,9E+09,9E+09]];
    CONST robtarget T437:=[[61.000031,74.473110,4.249591],[1.000000,0.000000,0.000000,0.000000],[0,0,-1,0],[9E+09,9E+09,9E+09,9E+09,9E+09,9E+09]];
    CONST robtarget T438:=[[62.500037,74.230221,4.249591],[1.000000,0.000000,0.000000,0.000000],[0,0,-1,0],[9E+09,9E+09,9E+09,9E+09,9E+09,9E+09]];
    CONST robtarget T439:=[[62.500037,37.641990,4.249591],[1.000000,0.000000,0.000000,0.000000],[0,0,-1,0],[9E+09,9E+09,9E+09,9E+09,9E+09,9E+09]];
    CONST robtarget T440:=[[64.000043,38.097323,4.249591],[1.000000,0.000000,0.000000,0.000000],[0,0,-1,0],[9E+09,9E+09,9E+09,9E+09,9E+09,9E+09]];
    CONST robtarget T441:=[[64.000043,73.715029,4.249591],[1.000000,0.000000,0.000000,0.000000],[0,0,-1,0],[9E+09,9E+09,9E+09,9E+09,9E+09,9E+09]];
    CONST robtarget T442:=[[65.500049,72.939577,4.249591],[1.000000,0.000000,0.000000,0.000000],[0,0,-1,0],[9E+09,9E+09,9E+09,9E+09,9E+09,9E+09]];
    CONST robtarget T443:=[[65.500049,38.592263,4.249591],[1.000000,0.000000,0.000000,0.000000],[0,0,-1,0],[9E+09,9E+09,9E+09,9E+09,9E+09,9E+09]];
    CONST robtarget T444:=[[67.000055,39.295226,4.249591],[1.000000,0.000000,0.000000,0.000000],[0,0,-1,0],[9E+09,9E+09,9E+09,9E+09,9E+09,9E+09]];
    CONST robtarget T445:=[[67.000055,71.924941,4.249591],[1.000000,0.000000,0.000000,0.000000],[0,0,-1,0],[9E+09,9E+09,9E+09,9E+09,9E+09,9E+09]];
    CONST robtarget T446:=[[68.500061,70.844693,4.249591],[1.000000,0.000000,0.000000,0.000000],[0,0,-1,0],[9E+09,9E+09,9E+09,9E+09,9E+09,9E+09]];
    CONST robtarget T447:=[[68.500061,40.066520,4.249591],[1.000000,0.000000,0.000000,0.000000],[0,0,-1,0],[9E+09,9E+09,9E+09,9E+09,9E+09,9E+09]];
    CONST robtarget T448:=[[70.000067,40.997440,4.249591],[1.000000,0.000000,0.000000,0.000000],[0,0,-1,0],[9E+09,9E+09,9E+09,9E+09,9E+09,9E+09]];
    CONST robtarget T449:=[[70.000067,69.500160,4.249591],[1.000000,0.000000,0.000000,0.000000],[0,0,-1,0],[9E+09,9E+09,9E+09,9E+09,9E+09,9E+09]];
    CONST robtarget T450:=[[71.500073,67.837825,4.249591],[1.000000,0.000000,0.000000,0.000000],[0,0,-1,0],[9E+09,9E+09,9E+09,9E+09,9E+09,9E+09]];
    CONST robtarget T451:=[[71.500073,42.013796,4.249591],[1.000000,0.000000,0.000000,0.000000],[0,0,-1,0],[9E+09,9E+09,9E+09,9E+09,9E+09,9E+09]];
    CONST robtarget T452:=[[73.000079,43.288408,4.249591],[1.000000,0.000000,0.000000,0.000000],[0,0,-1,0],[9E+09,9E+09,9E+09,9E+09,9E+09,9E+09]];
    CONST robtarget T453:=[[73.000079,65.775097,4.249591],[1.000000,0.000000,0.000000,0.000000],[0,0,-1,0],[9E+09,9E+09,9E+09,9E+09,9E+09,9E+09]];
    CONST robtarget T454:=[[74.500085,62.119811,4.249591],[1.000000,0.000000,0.000000,0.000000],[0,0,-1,0],[9E+09,9E+09,9E+09,9E+09,9E+09,9E+09]];
    CONST robtarget T455:=[[74.500085,44.766401,4.249591],[1.000000,0.000000,0.000000,0.000000],[0,0,-1,0],[9E+09,9E+09,9E+09,9E+09,9E+09,9E+09]];
    CONST robtarget T456:=[[76.000091,47.259741,4.249591],[1.000000,0.000000,0.000000,0.000000],[0,0,-1,0],[9E+09,9E+09,9E+09,9E+09,9E+09,9E+09]];
    CONST robtarget T457:=[[76.000091,56.726884,4.249591],[1.000000,0.000000,0.000000,0.000000],[0,0,-1,0],[9E+09,9E+09,9E+09,9E+09,9E+09,9E+09]];
    CONST robtarget T458:=[[76.000092,46.203974,4.749601],[1.000000,0.000000,0.000000,0.000000],[0,0,-1,0],[9E+09,9E+09,9E+09,9E+09,9E+09,9E+09]];
    CONST robtarget T459:=[[76.000092,58.050814,4.749601],[1.000000,0.000000,0.000000,0.000000],[0,0,-1,0],[9E+09,9E+09,9E+09,9E+09,9E+09,9E+09]];
    CONST robtarget T460:=[[76.000092,46.203974,4.749601],[1.000000,0.000000,0.000000,0.000000],[0,0,-1,0],[9E+09,9E+09,9E+09,9E+09,9E+09,9E+09]];
    CONST robtarget T461:=[[76.000092,58.050814,4.749601],[1.000000,0.000000,0.000000,0.000000],[0,0,-1,0],[9E+09,9E+09,9E+09,9E+09,9E+09,9E+09]];
    CONST robtarget T462:=[[74.500086,62.952276,4.749601],[1.000000,0.000000,0.000000,0.000000],[0,0,-1,0],[9E+09,9E+09,9E+09,9E+09,9E+09,9E+09]];
    CONST robtarget T463:=[[74.500086,44.133098,4.749601],[1.000000,0.000000,0.000000,0.000000],[0,0,-1,0],[9E+09,9E+09,9E+09,9E+09,9E+09,9E+09]];
    CONST robtarget T464:=[[73.000080,42.633630,4.749601],[1.000000,0.000000,0.000000,0.000000],[0,0,-1,0],[9E+09,9E+09,9E+09,9E+09,9E+09,9E+09]];
    CONST robtarget T465:=[[73.000080,66.117886,4.749601],[1.000000,0.000000,0.000000,0.000000],[0,0,-1,0],[9E+09,9E+09,9E+09,9E+09,9E+09,9E+09]];
    CONST robtarget T466:=[[71.500074,68.206758,4.749601],[1.000000,0.000000,0.000000,0.000000],[0,0,-1,0],[9E+09,9E+09,9E+09,9E+09,9E+09,9E+09]];
    CONST robtarget T467:=[[71.500074,41.435429,4.749601],[1.000000,0.000000,0.000000,0.000000],[0,0,-1,0],[9E+09,9E+09,9E+09,9E+09,9E+09,9E+09]];
    CONST robtarget T468:=[[70.000068,40.419825,4.749601],[1.000000,0.000000,0.000000,0.000000],[0,0,-1,0],[9E+09,9E+09,9E+09,9E+09,9E+09,9E+09]];
    CONST robtarget T469:=[[70.000068,69.854958,4.749601],[1.000000,0.000000,0.000000,0.000000],[0,0,-1,0],[9E+09,9E+09,9E+09,9E+09,9E+09,9E+09]];
    CONST robtarget T470:=[[68.500062,71.173927,4.749601],[1.000000,0.000000,0.000000,0.000000],[0,0,-1,0],[9E+09,9E+09,9E+09,9E+09,9E+09,9E+09]];
    CONST robtarget T471:=[[68.500062,39.460915,4.749601],[1.000000,0.000000,0.000000,0.000000],[0,0,-1,0],[9E+09,9E+09,9E+09,9E+09,9E+09,9E+09]];
    CONST robtarget T472:=[[67.000056,38.682860,4.749601],[1.000000,0.000000,0.000000,0.000000],[0,0,-1,0],[9E+09,9E+09,9E+09,9E+09,9E+09,9E+09]];
    CONST robtarget T473:=[[67.000056,72.341007,4.749601],[1.000000,0.000000,0.000000,0.000000],[0,0,-1,0],[9E+09,9E+09,9E+09,9E+09,9E+09,9E+09]];
    CONST robtarget T474:=[[65.500050,73.354303,4.749601],[1.000000,0.000000,0.000000,0.000000],[0,0,-1,0],[9E+09,9E+09,9E+09,9E+09,9E+09,9E+09]];
    CONST robtarget T475:=[[65.500050,37.962386,4.749601],[1.000000,0.000000,0.000000,0.000000],[0,0,-1,0],[9E+09,9E+09,9E+09,9E+09,9E+09,9E+09]];
    CONST robtarget T476:=[[64.000044,37.484916,4.749601],[1.000000,0.000000,0.000000,0.000000],[0,0,-1,0],[9E+09,9E+09,9E+09,9E+09,9E+09,9E+09]];
    CONST robtarget T477:=[[64.000044,74.123829,4.749601],[1.000000,0.000000,0.000000,0.000000],[0,0,-1,0],[9E+09,9E+09,9E+09,9E+09,9E+09,9E+09]];
    CONST robtarget T478:=[[62.500038,74.672381,4.749601],[1.000000,0.000000,0.000000,0.000000],[0,0,-1,0],[9E+09,9E+09,9E+09,9E+09,9E+09,9E+09]];
    CONST robtarget T479:=[[62.500038,37.078703,4.749601],[1.000000,0.000000,0.000000,0.000000],[0,0,-1,0],[9E+09,9E+09,9E+09,9E+09,9E+09,9E+09]];
    CONST robtarget T480:=[[61.000032,36.836181,4.749601],[1.000000,0.000000,0.000000,0.000000],[0,0,-1,0],[9E+09,9E+09,9E+09,9E+09,9E+09,9E+09]];
    CONST robtarget T481:=[[61.000032,74.928672,4.749601],[1.000000,0.000000,0.000000,0.000000],[0,0,-1,0],[9E+09,9E+09,9E+09,9E+09,9E+09,9E+09]];
    CONST robtarget T482:=[[59.500026,75.106604,4.749601],[1.000000,0.000000,0.000000,0.000000],[0,0,-1,0],[9E+09,9E+09,9E+09,9E+09,9E+09,9E+09]];
    CONST robtarget T483:=[[59.500026,36.627001,4.749601],[1.000000,0.000000,0.000000,0.000000],[0,0,-1,0],[9E+09,9E+09,9E+09,9E+09,9E+09,9E+09]];
    CONST robtarget T484:=[[58.000020,36.529364,4.749601],[1.000000,0.000000,0.000000,0.000000],[0,0,-1,0],[9E+09,9E+09,9E+09,9E+09,9E+09,9E+09]];
    CONST robtarget T485:=[[58.000020,75.195382,4.749601],[1.000000,0.000000,0.000000,0.000000],[0,0,-1,0],[9E+09,9E+09,9E+09,9E+09,9E+09,9E+09]];
    CONST robtarget T486:=[[56.500014,75.308911,4.749601],[1.000000,0.000000,0.000000,0.000000],[0,0,-1,0],[9E+09,9E+09,9E+09,9E+09,9E+09,9E+09]];
    CONST robtarget T487:=[[56.500014,36.485548,4.749601],[1.000000,0.000000,0.000000,0.000000],[0,0,-1,0],[9E+09,9E+09,9E+09,9E+09,9E+09,9E+09]];
    CONST robtarget T488:=[[55.000008,36.490372,4.749601],[1.000000,0.000000,0.000000,0.000000],[0,0,-1,0],[9E+09,9E+09,9E+09,9E+09,9E+09,9E+09]];
    CONST robtarget T489:=[[55.000008,75.392646,4.749601],[1.000000,0.000000,0.000000,0.000000],[0,0,-1,0],[9E+09,9E+09,9E+09,9E+09,9E+09,9E+09]];
    CONST robtarget T490:=[[53.500002,75.308911,4.749601],[1.000000,0.000000,0.000000,0.000000],[0,0,-1,0],[9E+09,9E+09,9E+09,9E+09,9E+09,9E+09]];
    CONST robtarget T491:=[[53.500002,36.485548,4.749601],[1.000000,0.000000,0.000000,0.000000],[0,0,-1,0],[9E+09,9E+09,9E+09,9E+09,9E+09,9E+09]];
    CONST robtarget T492:=[[51.999996,36.529364,4.749601],[1.000000,0.000000,0.000000,0.000000],[0,0,-1,0],[9E+09,9E+09,9E+09,9E+09,9E+09,9E+09]];
    CONST robtarget T493:=[[51.999996,75.195382,4.749601],[1.000000,0.000000,0.000000,0.000000],[0,0,-1,0],[9E+09,9E+09,9E+09,9E+09,9E+09,9E+09]];
    CONST robtarget T494:=[[50.499990,75.106604,4.749601],[1.000000,0.000000,0.000000,0.000000],[0,0,-1,0],[9E+09,9E+09,9E+09,9E+09,9E+09,9E+09]];
    CONST robtarget T495:=[[50.499990,36.627001,4.749601],[1.000000,0.000000,0.000000,0.000000],[0,0,-1,0],[9E+09,9E+09,9E+09,9E+09,9E+09,9E+09]];
    CONST robtarget T496:=[[48.999984,36.836181,4.749601],[1.000000,0.000000,0.000000,0.000000],[0,0,-1,0],[9E+09,9E+09,9E+09,9E+09,9E+09,9E+09]];
    CONST robtarget T497:=[[48.999984,74.928670,4.749601],[1.000000,0.000000,0.000000,0.000000],[0,0,-1,0],[9E+09,9E+09,9E+09,9E+09,9E+09,9E+09]];
    CONST robtarget T498:=[[47.499978,74.672375,4.749601],[1.000000,0.000000,0.000000,0.000000],[0,0,-1,0],[9E+09,9E+09,9E+09,9E+09,9E+09,9E+09]];
    CONST robtarget T499:=[[47.499978,37.078703,4.749601],[1.000000,0.000000,0.000000,0.000000],[0,0,-1,0],[9E+09,9E+09,9E+09,9E+09,9E+09,9E+09]];
    CONST robtarget T500:=[[45.999972,37.484916,4.749601],[1.000000,0.000000,0.000000,0.000000],[0,0,-1,0],[9E+09,9E+09,9E+09,9E+09,9E+09,9E+09]];
    CONST robtarget T501:=[[45.999972,74.123821,4.749601],[1.000000,0.000000,0.000000,0.000000],[0,0,-1,0],[9E+09,9E+09,9E+09,9E+09,9E+09,9E+09]];
    CONST robtarget T502:=[[44.499966,73.354295,4.749601],[1.000000,0.000000,0.000000,0.000000],[0,0,-1,0],[9E+09,9E+09,9E+09,9E+09,9E+09,9E+09]];
    CONST robtarget T503:=[[44.499966,37.962387,4.749601],[1.000000,0.000000,0.000000,0.000000],[0,0,-1,0],[9E+09,9E+09,9E+09,9E+09,9E+09,9E+09]];
    CONST robtarget T504:=[[42.999960,38.682860,4.749601],[1.000000,0.000000,0.000000,0.000000],[0,0,-1,0],[9E+09,9E+09,9E+09,9E+09,9E+09,9E+09]];
    CONST robtarget T505:=[[42.999960,72.341006,4.749601],[1.000000,0.000000,0.000000,0.000000],[0,0,-1,0],[9E+09,9E+09,9E+09,9E+09,9E+09,9E+09]];
    CONST robtarget T506:=[[41.499954,71.173928,4.749601],[1.000000,0.000000,0.000000,0.000000],[0,0,-1,0],[9E+09,9E+09,9E+09,9E+09,9E+09,9E+09]];
    CONST robtarget T507:=[[41.499954,39.460914,4.749601],[1.000000,0.000000,0.000000,0.000000],[0,0,-1,0],[9E+09,9E+09,9E+09,9E+09,9E+09,9E+09]];
    CONST robtarget T508:=[[39.999948,40.419824,4.749601],[1.000000,0.000000,0.000000,0.000000],[0,0,-1,0],[9E+09,9E+09,9E+09,9E+09,9E+09,9E+09]];
    CONST robtarget T509:=[[39.999948,69.854959,4.749601],[1.000000,0.000000,0.000000,0.000000],[0,0,-1,0],[9E+09,9E+09,9E+09,9E+09,9E+09,9E+09]];
    CONST robtarget T510:=[[38.499942,68.206764,4.749601],[1.000000,0.000000,0.000000,0.000000],[0,0,-1,0],[9E+09,9E+09,9E+09,9E+09,9E+09,9E+09]];
    CONST robtarget T511:=[[38.499942,41.435428,4.749601],[1.000000,0.000000,0.000000,0.000000],[0,0,-1,0],[9E+09,9E+09,9E+09,9E+09,9E+09,9E+09]];
    CONST robtarget T512:=[[36.999936,42.633629,4.749601],[1.000000,0.000000,0.000000,0.000000],[0,0,-1,0],[9E+09,9E+09,9E+09,9E+09,9E+09,9E+09]];
    CONST robtarget T513:=[[36.999936,66.120190,4.749601],[1.000000,0.000000,0.000000,0.000000],[0,0,-1,0],[9E+09,9E+09,9E+09,9E+09,9E+09,9E+09]];
    CONST robtarget T514:=[[35.499930,62.972222,4.749601],[1.000000,0.000000,0.000000,0.000000],[0,0,-1,0],[9E+09,9E+09,9E+09,9E+09,9E+09,9E+09]];
    CONST robtarget T515:=[[35.499930,44.133096,4.749601],[1.000000,0.000000,0.000000,0.000000],[0,0,-1,0],[9E+09,9E+09,9E+09,9E+09,9E+09,9E+09]];
    CONST robtarget T516:=[[33.999924,46.203970,4.749601],[1.000000,0.000000,0.000000,0.000000],[0,0,-1,0],[9E+09,9E+09,9E+09,9E+09,9E+09,9E+09]];
    CONST robtarget T517:=[[33.999924,58.076657,4.749601],[1.000000,0.000000,0.000000,0.000000],[0,0,-1,0],[9E+09,9E+09,9E+09,9E+09,9E+09,9E+09]];
    CONST robtarget T518:=[[33.249920,46.763494,5.249611],[1.000000,0.000000,0.000000,0.000000],[0,0,-1,0],[9E+09,9E+09,9E+09,9E+09,9E+09,9E+09]];
    CONST robtarget T519:=[[33.249920,55.860723,5.249611],[1.000000,0.000000,0.000000,0.000000],[0,0,-1,0],[9E+09,9E+09,9E+09,9E+09,9E+09,9E+09]];
    CONST robtarget T520:=[[33.249920,46.763494,5.249611],[1.000000,0.000000,0.000000,0.000000],[0,0,-1,0],[9E+09,9E+09,9E+09,9E+09,9E+09,9E+09]];
    CONST robtarget T521:=[[33.249920,55.860723,5.249611],[1.000000,0.000000,0.000000,0.000000],[0,0,-1,0],[9E+09,9E+09,9E+09,9E+09,9E+09,9E+09]];
    CONST robtarget T522:=[[34.749926,61.294733,5.249611],[1.000000,0.000000,0.000000,0.000000],[0,0,-1,0],[9E+09,9E+09,9E+09,9E+09,9E+09,9E+09]];
    CONST robtarget T523:=[[34.749926,44.245212,5.249611],[1.000000,0.000000,0.000000,0.000000],[0,0,-1,0],[9E+09,9E+09,9E+09,9E+09,9E+09,9E+09]];
    CONST robtarget T524:=[[36.249932,42.728584,5.249611],[1.000000,0.000000,0.000000,0.000000],[0,0,-1,0],[9E+09,9E+09,9E+09,9E+09,9E+09,9E+09]];
    CONST robtarget T525:=[[36.249932,65.233359,5.249611],[1.000000,0.000000,0.000000,0.000000],[0,0,-1,0],[9E+09,9E+09,9E+09,9E+09,9E+09,9E+09]];
    CONST robtarget T526:=[[37.749938,67.527018,5.249611],[1.000000,0.000000,0.000000,0.000000],[0,0,-1,0],[9E+09,9E+09,9E+09,9E+09,9E+09,9E+09]];
    CONST robtarget T527:=[[37.749938,41.448496,5.249611],[1.000000,0.000000,0.000000,0.000000],[0,0,-1,0],[9E+09,9E+09,9E+09,9E+09,9E+09,9E+09]];
    CONST robtarget T528:=[[39.249944,40.287239,5.249611],[1.000000,0.000000,0.000000,0.000000],[0,0,-1,0],[9E+09,9E+09,9E+09,9E+09,9E+09,9E+09]];
    CONST robtarget T529:=[[39.249944,69.393900,5.249611],[1.000000,0.000000,0.000000,0.000000],[0,0,-1,0],[9E+09,9E+09,9E+09,9E+09,9E+09,9E+09]];
    CONST robtarget T530:=[[40.749950,70.881736,5.249611],[1.000000,0.000000,0.000000,0.000000],[0,0,-1,0],[9E+09,9E+09,9E+09,9E+09,9E+09,9E+09]];
    CONST robtarget T531:=[[40.749950,39.336086,5.249611],[1.000000,0.000000,0.000000,0.000000],[0,0,-1,0],[9E+09,9E+09,9E+09,9E+09,9E+09,9E+09]];
    CONST robtarget T532:=[[42.249956,38.432409,5.249611],[1.000000,0.000000,0.000000,0.000000],[0,0,-1,0],[9E+09,9E+09,9E+09,9E+09,9E+09,9E+09]];
    CONST robtarget T533:=[[42.249956,72.177277,5.249611],[1.000000,0.000000,0.000000,0.000000],[0,0,-1,0],[9E+09,9E+09,9E+09,9E+09,9E+09,9E+09]];
    CONST robtarget T534:=[[43.749962,73.236198,5.249611],[1.000000,0.000000,0.000000,0.000000],[0,0,-1,0],[9E+09,9E+09,9E+09,9E+09,9E+09,9E+09]];
    CONST robtarget T535:=[[43.749962,37.783096,5.249611],[1.000000,0.000000,0.000000,0.000000],[0,0,-1,0],[9E+09,9E+09,9E+09,9E+09,9E+09,9E+09]];
    CONST robtarget T536:=[[45.249968,37.257265,5.249611],[1.000000,0.000000,0.000000,0.000000],[0,0,-1,0],[9E+09,9E+09,9E+09,9E+09,9E+09,9E+09]];
    CONST robtarget T537:=[[45.249968,74.180372,5.249611],[1.000000,0.000000,0.000000,0.000000],[0,0,-1,0],[9E+09,9E+09,9E+09,9E+09,9E+09,9E+09]];
    CONST robtarget T538:=[[46.749974,74.882582,5.249611],[1.000000,0.000000,0.000000,0.000000],[0,0,-1,0],[9E+09,9E+09,9E+09,9E+09,9E+09,9E+09]];
    CONST robtarget T539:=[[46.749974,36.856340,5.249611],[1.000000,0.000000,0.000000,0.000000],[0,0,-1,0],[9E+09,9E+09,9E+09,9E+09,9E+09,9E+09]];
    CONST robtarget T540:=[[48.249980,36.540907,5.249611],[1.000000,0.000000,0.000000,0.000000],[0,0,-1,0],[9E+09,9E+09,9E+09,9E+09,9E+09,9E+09]];
    CONST robtarget T541:=[[48.249980,75.245971,5.249611],[1.000000,0.000000,0.000000,0.000000],[0,0,-1,0],[9E+09,9E+09,9E+09,9E+09,9E+09,9E+09]];
    CONST robtarget T542:=[[49.749986,75.515166,5.249611],[1.000000,0.000000,0.000000,0.000000],[0,0,-1,0],[9E+09,9E+09,9E+09,9E+09,9E+09,9E+09]];
    CONST robtarget T543:=[[49.749986,36.307129,5.249611],[1.000000,0.000000,0.000000,0.000000],[0,0,-1,0],[9E+09,9E+09,9E+09,9E+09,9E+09,9E+09]];
    CONST robtarget T544:=[[51.249992,36.203811,5.249611],[1.000000,0.000000,0.000000,0.000000],[0,0,-1,0],[9E+09,9E+09,9E+09,9E+09,9E+09,9E+09]];
    CONST robtarget T545:=[[51.249992,75.627007,5.249611],[1.000000,0.000000,0.000000,0.000000],[0,0,-1,0],[9E+09,9E+09,9E+09,9E+09,9E+09,9E+09]];
    CONST robtarget T546:=[[52.749998,75.734929,5.249611],[1.000000,0.000000,0.000000,0.000000],[0,0,-1,0],[9E+09,9E+09,9E+09,9E+09,9E+09,9E+09]];
    CONST robtarget T547:=[[52.749998,36.110049,5.249611],[1.000000,0.000000,0.000000,0.000000],[0,0,-1,0],[9E+09,9E+09,9E+09,9E+09,9E+09,9E+09]];
    CONST robtarget T548:=[[54.250004,36.114911,5.249611],[1.000000,0.000000,0.000000,0.000000],[0,0,-1,0],[9E+09,9E+09,9E+09,9E+09,9E+09,9E+09]];
    CONST robtarget T549:=[[54.250004,75.858380,5.249611],[1.000000,0.000000,0.000000,0.000000],[0,0,-1,0],[9E+09,9E+09,9E+09,9E+09,9E+09,9E+09]];
    CONST robtarget T550:=[[55.750010,75.858380,5.249611],[1.000000,0.000000,0.000000,0.000000],[0,0,-1,0],[9E+09,9E+09,9E+09,9E+09,9E+09,9E+09]];
    CONST robtarget T551:=[[55.750010,36.114911,5.249611],[1.000000,0.000000,0.000000,0.000000],[0,0,-1,0],[9E+09,9E+09,9E+09,9E+09,9E+09,9E+09]];
    CONST robtarget T552:=[[57.250016,36.110049,5.249611],[1.000000,0.000000,0.000000,0.000000],[0,0,-1,0],[9E+09,9E+09,9E+09,9E+09,9E+09,9E+09]];
    CONST robtarget T553:=[[57.250016,75.734929,5.249611],[1.000000,0.000000,0.000000,0.000000],[0,0,-1,0],[9E+09,9E+09,9E+09,9E+09,9E+09,9E+09]];
    CONST robtarget T554:=[[58.750022,75.627007,5.249611],[1.000000,0.000000,0.000000,0.000000],[0,0,-1,0],[9E+09,9E+09,9E+09,9E+09,9E+09,9E+09]];
    CONST robtarget T555:=[[58.750022,36.203811,5.249611],[1.000000,0.000000,0.000000,0.000000],[0,0,-1,0],[9E+09,9E+09,9E+09,9E+09,9E+09,9E+09]];
    CONST robtarget T556:=[[60.250028,36.307129,5.249611],[1.000000,0.000000,0.000000,0.000000],[0,0,-1,0],[9E+09,9E+09,9E+09,9E+09,9E+09,9E+09]];
    CONST robtarget T557:=[[60.250028,75.515165,5.249611],[1.000000,0.000000,0.000000,0.000000],[0,0,-1,0],[9E+09,9E+09,9E+09,9E+09,9E+09,9E+09]];
    CONST robtarget T558:=[[61.750034,75.245978,5.249611],[1.000000,0.000000,0.000000,0.000000],[0,0,-1,0],[9E+09,9E+09,9E+09,9E+09,9E+09,9E+09]];
    CONST robtarget T559:=[[61.750034,36.540907,5.249611],[1.000000,0.000000,0.000000,0.000000],[0,0,-1,0],[9E+09,9E+09,9E+09,9E+09,9E+09,9E+09]];
    CONST robtarget T560:=[[63.250040,36.856340,5.249611],[1.000000,0.000000,0.000000,0.000000],[0,0,-1,0],[9E+09,9E+09,9E+09,9E+09,9E+09,9E+09]];
    CONST robtarget T561:=[[63.250040,74.882592,5.249611],[1.000000,0.000000,0.000000,0.000000],[0,0,-1,0],[9E+09,9E+09,9E+09,9E+09,9E+09,9E+09]];
    CONST robtarget T562:=[[64.750046,74.180380,5.249611],[1.000000,0.000000,0.000000,0.000000],[0,0,-1,0],[9E+09,9E+09,9E+09,9E+09,9E+09,9E+09]];
    CONST robtarget T563:=[[64.750046,37.257265,5.249611],[1.000000,0.000000,0.000000,0.000000],[0,0,-1,0],[9E+09,9E+09,9E+09,9E+09,9E+09,9E+09]];
    CONST robtarget T564:=[[66.250052,37.783096,5.249611],[1.000000,0.000000,0.000000,0.000000],[0,0,-1,0],[9E+09,9E+09,9E+09,9E+09,9E+09,9E+09]];
    CONST robtarget T565:=[[66.250052,73.236200,5.249611],[1.000000,0.000000,0.000000,0.000000],[0,0,-1,0],[9E+09,9E+09,9E+09,9E+09,9E+09,9E+09]];
    CONST robtarget T566:=[[67.750058,72.177277,5.249611],[1.000000,0.000000,0.000000,0.000000],[0,0,-1,0],[9E+09,9E+09,9E+09,9E+09,9E+09,9E+09]];
    CONST robtarget T567:=[[67.750058,38.432409,5.249611],[1.000000,0.000000,0.000000,0.000000],[0,0,-1,0],[9E+09,9E+09,9E+09,9E+09,9E+09,9E+09]];
    CONST robtarget T568:=[[69.250064,39.336087,5.249611],[1.000000,0.000000,0.000000,0.000000],[0,0,-1,0],[9E+09,9E+09,9E+09,9E+09,9E+09,9E+09]];
    CONST robtarget T569:=[[69.250064,70.881735,5.249611],[1.000000,0.000000,0.000000,0.000000],[0,0,-1,0],[9E+09,9E+09,9E+09,9E+09,9E+09,9E+09]];
    CONST robtarget T570:=[[70.750070,69.393898,5.249611],[1.000000,0.000000,0.000000,0.000000],[0,0,-1,0],[9E+09,9E+09,9E+09,9E+09,9E+09,9E+09]];
    CONST robtarget T571:=[[70.750070,40.287240,5.249611],[1.000000,0.000000,0.000000,0.000000],[0,0,-1,0],[9E+09,9E+09,9E+09,9E+09,9E+09,9E+09]];
    CONST robtarget T572:=[[72.250076,41.448498,5.249611],[1.000000,0.000000,0.000000,0.000000],[0,0,-1,0],[9E+09,9E+09,9E+09,9E+09,9E+09,9E+09]];
    CONST robtarget T573:=[[72.250076,67.526203,5.249611],[1.000000,0.000000,0.000000,0.000000],[0,0,-1,0],[9E+09,9E+09,9E+09,9E+09,9E+09,9E+09]];
    CONST robtarget T574:=[[73.750082,65.227528,5.249611],[1.000000,0.000000,0.000000,0.000000],[0,0,-1,0],[9E+09,9E+09,9E+09,9E+09,9E+09,9E+09]];
    CONST robtarget T575:=[[73.750082,42.728585,5.249611],[1.000000,0.000000,0.000000,0.000000],[0,0,-1,0],[9E+09,9E+09,9E+09,9E+09,9E+09,9E+09]];
    CONST robtarget T576:=[[75.250088,44.245214,5.249611],[1.000000,0.000000,0.000000,0.000000],[0,0,-1,0],[9E+09,9E+09,9E+09,9E+09,9E+09,9E+09]];
    CONST robtarget T577:=[[75.250088,61.262516,5.249611],[1.000000,0.000000,0.000000,0.000000],[0,0,-1,0],[9E+09,9E+09,9E+09,9E+09,9E+09,9E+09]];
    CONST robtarget T578:=[[76.750094,55.847932,5.249611],[1.000000,0.000000,0.000000,0.000000],[0,0,-1,0],[9E+09,9E+09,9E+09,9E+09,9E+09,9E+09]];
    CONST robtarget T579:=[[76.750094,46.763502,5.249611],[1.000000,0.000000,0.000000,0.000000],[0,0,-1,0],[9E+09,9E+09,9E+09,9E+09,9E+09,9E+09]];
    CONST robtarget T580:=[[76.750094,46.148766,5.749621],[1.000000,0.000000,0.000000,0.000000],[0,0,-1,0],[9E+09,9E+09,9E+09,9E+09,9E+09,9E+09]];
    CONST robtarget T581:=[[76.750094,56.999042,5.749621],[1.000000,0.000000,0.000000,0.000000],[0,0,-1,0],[9E+09,9E+09,9E+09,9E+09,9E+09,9E+09]];
    CONST robtarget T582:=[[76.750094,46.148766,5.749621],[1.000000,0.000000,0.000000,0.000000],[0,0,-1,0],[9E+09,9E+09,9E+09,9E+09,9E+09,9E+09]];
    CONST robtarget T583:=[[76.750094,56.999042,5.749621],[1.000000,0.000000,0.000000,0.000000],[0,0,-1,0],[9E+09,9E+09,9E+09,9E+09,9E+09,9E+09]];
    CONST robtarget T584:=[[75.250088,61.857288,5.749621],[1.000000,0.000000,0.000000,0.000000],[0,0,-1,0],[9E+09,9E+09,9E+09,9E+09,9E+09,9E+09]];
    CONST robtarget T585:=[[75.250088,43.769918,5.749621],[1.000000,0.000000,0.000000,0.000000],[0,0,-1,0],[9E+09,9E+09,9E+09,9E+09,9E+09,9E+09]];
    CONST robtarget T586:=[[73.750082,42.169937,5.749621],[1.000000,0.000000,0.000000,0.000000],[0,0,-1,0],[9E+09,9E+09,9E+09,9E+09,9E+09,9E+09]];
    CONST robtarget T587:=[[73.750082,65.640558,5.749621],[1.000000,0.000000,0.000000,0.000000],[0,0,-1,0],[9E+09,9E+09,9E+09,9E+09,9E+09,9E+09]];
    CONST robtarget T588:=[[72.250076,67.895137,5.749621],[1.000000,0.000000,0.000000,0.000000],[0,0,-1,0],[9E+09,9E+09,9E+09,9E+09,9E+09,9E+09]];
    CONST robtarget T589:=[[72.250076,40.937334,5.749621],[1.000000,0.000000,0.000000,0.000000],[0,0,-1,0],[9E+09,9E+09,9E+09,9E+09,9E+09,9E+09]];
    CONST robtarget T590:=[[70.750070,39.761045,5.749621],[1.000000,0.000000,0.000000,0.000000],[0,0,-1,0],[9E+09,9E+09,9E+09,9E+09,9E+09,9E+09]];
    CONST robtarget T591:=[[70.750070,69.716607,5.749621],[1.000000,0.000000,0.000000,0.000000],[0,0,-1,0],[9E+09,9E+09,9E+09,9E+09,9E+09,9E+09]];
    CONST robtarget T592:=[[69.250064,71.222870,5.749621],[1.000000,0.000000,0.000000,0.000000],[0,0,-1,0],[9E+09,9E+09,9E+09,9E+09,9E+09,9E+09]];
    CONST robtarget T593:=[[69.250064,38.830794,5.749621],[1.000000,0.000000,0.000000,0.000000],[0,0,-1,0],[9E+09,9E+09,9E+09,9E+09,9E+09,9E+09]];
    CONST robtarget T594:=[[67.750058,37.987251,5.749621],[1.000000,0.000000,0.000000,0.000000],[0,0,-1,0],[9E+09,9E+09,9E+09,9E+09,9E+09,9E+09]];
    CONST robtarget T595:=[[67.750058,72.538760,5.749621],[1.000000,0.000000,0.000000,0.000000],[0,0,-1,0],[9E+09,9E+09,9E+09,9E+09,9E+09,9E+09]];
    CONST robtarget T596:=[[66.250052,73.604088,5.749621],[1.000000,0.000000,0.000000,0.000000],[0,0,-1,0],[9E+09,9E+09,9E+09,9E+09,9E+09,9E+09]];
    CONST robtarget T597:=[[66.250052,37.342352,5.749621],[1.000000,0.000000,0.000000,0.000000],[0,0,-1,0],[9E+09,9E+09,9E+09,9E+09,9E+09,9E+09]];
    CONST robtarget T598:=[[64.750046,36.828601,5.749621],[1.000000,0.000000,0.000000,0.000000],[0,0,-1,0],[9E+09,9E+09,9E+09,9E+09,9E+09,9E+09]];
    CONST robtarget T599:=[[64.750046,74.586660,5.749621],[1.000000,0.000000,0.000000,0.000000],[0,0,-1,0],[9E+09,9E+09,9E+09,9E+09,9E+09,9E+09]];
    CONST robtarget T600:=[[63.250040,75.290269,5.749621],[1.000000,0.000000,0.000000,0.000000],[0,0,-1,0],[9E+09,9E+09,9E+09,9E+09,9E+09,9E+09]];
    CONST robtarget T601:=[[63.250040,36.435933,5.749621],[1.000000,0.000000,0.000000,0.000000],[0,0,-1,0],[9E+09,9E+09,9E+09,9E+09,9E+09,9E+09]];
    CONST robtarget T602:=[[61.750034,36.124372,5.749621],[1.000000,0.000000,0.000000,0.000000],[0,0,-1,0],[9E+09,9E+09,9E+09,9E+09,9E+09,9E+09]];
    CONST robtarget T603:=[[61.750034,75.673914,5.749621],[1.000000,0.000000,0.000000,0.000000],[0,0,-1,0],[9E+09,9E+09,9E+09,9E+09,9E+09,9E+09]];
    CONST robtarget T604:=[[60.250028,75.905471,5.749621],[1.000000,0.000000,0.000000,0.000000],[0,0,-1,0],[9E+09,9E+09,9E+09,9E+09,9E+09,9E+09]];
    CONST robtarget T605:=[[60.250028,35.919583,5.749621],[1.000000,0.000000,0.000000,0.000000],[0,0,-1,0],[9E+09,9E+09,9E+09,9E+09,9E+09,9E+09]];
    CONST robtarget T606:=[[58.750022,35.829359,5.749621],[1.000000,0.000000,0.000000,0.000000],[0,0,-1,0],[9E+09,9E+09,9E+09,9E+09,9E+09,9E+09]];
    CONST robtarget T607:=[[58.750022,76.015573,5.749621],[1.000000,0.000000,0.000000,0.000000],[0,0,-1,0],[9E+09,9E+09,9E+09,9E+09,9E+09,9E+09]];
    CONST robtarget T608:=[[57.250016,76.146335,5.749621],[1.000000,0.000000,0.000000,0.000000],[0,0,-1,0],[9E+09,9E+09,9E+09,9E+09,9E+09,9E+09]];
    CONST robtarget T609:=[[57.250016,35.736982,5.749621],[1.000000,0.000000,0.000000,0.000000],[0,0,-1,0],[9E+09,9E+09,9E+09,9E+09,9E+09,9E+09]];
    CONST robtarget T610:=[[55.750010,35.741756,5.749621],[1.000000,0.000000,0.000000,0.000000],[0,0,-1,0],[9E+09,9E+09,9E+09,9E+09,9E+09,9E+09]];
    CONST robtarget T611:=[[55.750010,76.267629,5.749621],[1.000000,0.000000,0.000000,0.000000],[0,0,-1,0],[9E+09,9E+09,9E+09,9E+09,9E+09,9E+09]];
    CONST robtarget T612:=[[54.250004,76.267629,5.749621],[1.000000,0.000000,0.000000,0.000000],[0,0,-1,0],[9E+09,9E+09,9E+09,9E+09,9E+09,9E+09]];
    CONST robtarget T613:=[[54.250004,35.741756,5.749621],[1.000000,0.000000,0.000000,0.000000],[0,0,-1,0],[9E+09,9E+09,9E+09,9E+09,9E+09,9E+09]];
    CONST robtarget T614:=[[52.749998,35.736982,5.749621],[1.000000,0.000000,0.000000,0.000000],[0,0,-1,0],[9E+09,9E+09,9E+09,9E+09,9E+09,9E+09]];
    CONST robtarget T615:=[[52.749998,76.146335,5.749621],[1.000000,0.000000,0.000000,0.000000],[0,0,-1,0],[9E+09,9E+09,9E+09,9E+09,9E+09,9E+09]];
    CONST robtarget T616:=[[51.249992,76.015573,5.749621],[1.000000,0.000000,0.000000,0.000000],[0,0,-1,0],[9E+09,9E+09,9E+09,9E+09,9E+09,9E+09]];
    CONST robtarget T617:=[[51.249992,35.829359,5.749621],[1.000000,0.000000,0.000000,0.000000],[0,0,-1,0],[9E+09,9E+09,9E+09,9E+09,9E+09,9E+09]];
    CONST robtarget T618:=[[49.749986,35.919583,5.749621],[1.000000,0.000000,0.000000,0.000000],[0,0,-1,0],[9E+09,9E+09,9E+09,9E+09,9E+09,9E+09]];
    CONST robtarget T619:=[[49.749986,75.905472,5.749621],[1.000000,0.000000,0.000000,0.000000],[0,0,-1,0],[9E+09,9E+09,9E+09,9E+09,9E+09,9E+09]];
    CONST robtarget T620:=[[48.249980,75.673906,5.749621],[1.000000,0.000000,0.000000,0.000000],[0,0,-1,0],[9E+09,9E+09,9E+09,9E+09,9E+09,9E+09]];
    CONST robtarget T621:=[[48.249980,36.124372,5.749621],[1.000000,0.000000,0.000000,0.000000],[0,0,-1,0],[9E+09,9E+09,9E+09,9E+09,9E+09,9E+09]];
    CONST robtarget T622:=[[46.749974,36.435933,5.749621],[1.000000,0.000000,0.000000,0.000000],[0,0,-1,0],[9E+09,9E+09,9E+09,9E+09,9E+09,9E+09]];
    CONST robtarget T623:=[[46.749974,75.290258,5.749621],[1.000000,0.000000,0.000000,0.000000],[0,0,-1,0],[9E+09,9E+09,9E+09,9E+09,9E+09,9E+09]];
    CONST robtarget T624:=[[45.249968,74.586656,5.749621],[1.000000,0.000000,0.000000,0.000000],[0,0,-1,0],[9E+09,9E+09,9E+09,9E+09,9E+09,9E+09]];
    CONST robtarget T625:=[[45.249968,36.828602,5.749621],[1.000000,0.000000,0.000000,0.000000],[0,0,-1,0],[9E+09,9E+09,9E+09,9E+09,9E+09,9E+09]];
    CONST robtarget T626:=[[43.749962,37.342353,5.749621],[1.000000,0.000000,0.000000,0.000000],[0,0,-1,0],[9E+09,9E+09,9E+09,9E+09,9E+09,9E+09]];
    CONST robtarget T627:=[[43.749962,73.604086,5.749621],[1.000000,0.000000,0.000000,0.000000],[0,0,-1,0],[9E+09,9E+09,9E+09,9E+09,9E+09,9E+09]];
    CONST robtarget T628:=[[42.249956,72.538760,5.749621],[1.000000,0.000000,0.000000,0.000000],[0,0,-1,0],[9E+09,9E+09,9E+09,9E+09,9E+09,9E+09]];
    CONST robtarget T629:=[[42.249956,37.987251,5.749621],[1.000000,0.000000,0.000000,0.000000],[0,0,-1,0],[9E+09,9E+09,9E+09,9E+09,9E+09,9E+09]];
    CONST robtarget T630:=[[40.749950,38.830794,5.749621],[1.000000,0.000000,0.000000,0.000000],[0,0,-1,0],[9E+09,9E+09,9E+09,9E+09,9E+09,9E+09]];
    CONST robtarget T631:=[[40.749950,71.222871,5.749621],[1.000000,0.000000,0.000000,0.000000],[0,0,-1,0],[9E+09,9E+09,9E+09,9E+09,9E+09,9E+09]];
    CONST robtarget T632:=[[39.249944,69.716607,5.749621],[1.000000,0.000000,0.000000,0.000000],[0,0,-1,0],[9E+09,9E+09,9E+09,9E+09,9E+09,9E+09]];
    CONST robtarget T633:=[[39.249944,39.761044,5.749621],[1.000000,0.000000,0.000000,0.000000],[0,0,-1,0],[9E+09,9E+09,9E+09,9E+09,9E+09,9E+09]];
    CONST robtarget T634:=[[37.749938,40.937333,5.749621],[1.000000,0.000000,0.000000,0.000000],[0,0,-1,0],[9E+09,9E+09,9E+09,9E+09,9E+09,9E+09]];
    CONST robtarget T635:=[[37.749938,67.895683,5.749621],[1.000000,0.000000,0.000000,0.000000],[0,0,-1,0],[9E+09,9E+09,9E+09,9E+09,9E+09,9E+09]];
    CONST robtarget T636:=[[36.249932,65.645088,5.749621],[1.000000,0.000000,0.000000,0.000000],[0,0,-1,0],[9E+09,9E+09,9E+09,9E+09,9E+09,9E+09]];
    CONST robtarget T637:=[[36.249932,42.169936,5.749621],[1.000000,0.000000,0.000000,0.000000],[0,0,-1,0],[9E+09,9E+09,9E+09,9E+09,9E+09,9E+09]];
    CONST robtarget T638:=[[34.749926,43.769917,5.749621],[1.000000,0.000000,0.000000,0.000000],[0,0,-1,0],[9E+09,9E+09,9E+09,9E+09,9E+09,9E+09]];
    CONST robtarget T639:=[[34.749926,61.884738,5.749621],[1.000000,0.000000,0.000000,0.000000],[0,0,-1,0],[9E+09,9E+09,9E+09,9E+09,9E+09,9E+09]];
    CONST robtarget T640:=[[33.249920,57.018167,5.749621],[1.000000,0.000000,0.000000,0.000000],[0,0,-1,0],[9E+09,9E+09,9E+09,9E+09,9E+09,9E+09]];
    CONST robtarget T641:=[[33.249920,46.148763,5.749621],[1.000000,0.000000,0.000000,0.000000],[0,0,-1,0],[9E+09,9E+09,9E+09,9E+09,9E+09,9E+09]];
    CONST robtarget T642:=[[32.499917,47.712287,6.249631],[1.000000,0.000000,0.000000,0.000000],[0,0,-1,0],[9E+09,9E+09,9E+09,9E+09,9E+09,9E+09]];
    CONST robtarget T643:=[[32.499917,54.842849,6.249631],[1.000000,0.000000,0.000000,0.000000],[0,0,-1,0],[9E+09,9E+09,9E+09,9E+09,9E+09,9E+09]];
    CONST robtarget T644:=[[32.499917,47.712287,6.249631],[1.000000,0.000000,0.000000,0.000000],[0,0,-1,0],[9E+09,9E+09,9E+09,9E+09,9E+09,9E+09]];
    CONST robtarget T645:=[[32.499917,54.842849,6.249631],[1.000000,0.000000,0.000000,0.000000],[0,0,-1,0],[9E+09,9E+09,9E+09,9E+09,9E+09,9E+09]];
    CONST robtarget T646:=[[33.999923,60.383683,6.249631],[1.000000,0.000000,0.000000,0.000000],[0,0,-1,0],[9E+09,9E+09,9E+09,9E+09,9E+09,9E+09]];
    CONST robtarget T647:=[[33.999923,44.225147,6.249631],[1.000000,0.000000,0.000000,0.000000],[0,0,-1,0],[9E+09,9E+09,9E+09,9E+09,9E+09,9E+09]];
    CONST robtarget T648:=[[35.499929,42.494021,6.249631],[1.000000,0.000000,0.000000,0.000000],[0,0,-1,0],[9E+09,9E+09,9E+09,9E+09,9E+09,9E+09]];
    CONST robtarget T649:=[[35.499929,64.397148,6.249631],[1.000000,0.000000,0.000000,0.000000],[0,0,-1,0],[9E+09,9E+09,9E+09,9E+09,9E+09,9E+09]];
    CONST robtarget T650:=[[36.999935,66.947484,6.249631],[1.000000,0.000000,0.000000,0.000000],[0,0,-1,0],[9E+09,9E+09,9E+09,9E+09,9E+09,9E+09]];
    CONST robtarget T651:=[[36.999935,41.103880,6.249631],[1.000000,0.000000,0.000000,0.000000],[0,0,-1,0],[9E+09,9E+09,9E+09,9E+09,9E+09,9E+09]];
    CONST robtarget T652:=[[38.499941,39.891105,6.249631],[1.000000,0.000000,0.000000,0.000000],[0,0,-1,0],[9E+09,9E+09,9E+09,9E+09,9E+09,9E+09]];
    CONST robtarget T653:=[[38.499941,69.078100,6.249631],[1.000000,0.000000,0.000000,0.000000],[0,0,-1,0],[9E+09,9E+09,9E+09,9E+09,9E+09,9E+09]];
    CONST robtarget T654:=[[39.999947,70.867703,6.249631],[1.000000,0.000000,0.000000,0.000000],[0,0,-1,0],[9E+09,9E+09,9E+09,9E+09,9E+09,9E+09]];
    CONST robtarget T655:=[[39.999947,38.836205,6.249631],[1.000000,0.000000,0.000000,0.000000],[0,0,-1,0],[9E+09,9E+09,9E+09,9E+09,9E+09,9E+09]];
    CONST robtarget T656:=[[41.499953,37.908305,6.249631],[1.000000,0.000000,0.000000,0.000000],[0,0,-1,0],[9E+09,9E+09,9E+09,9E+09,9E+09,9E+09]];
    CONST robtarget T657:=[[41.499953,72.303443,6.249631],[1.000000,0.000000,0.000000,0.000000],[0,0,-1,0],[9E+09,9E+09,9E+09,9E+09,9E+09,9E+09]];
    CONST robtarget T658:=[[42.999959,73.456701,6.249631],[1.000000,0.000000,0.000000,0.000000],[0,0,-1,0],[9E+09,9E+09,9E+09,9E+09,9E+09,9E+09]];
    CONST robtarget T659:=[[42.999959,37.225943,6.249631],[1.000000,0.000000,0.000000,0.000000],[0,0,-1,0],[9E+09,9E+09,9E+09,9E+09,9E+09,9E+09]];
    CONST robtarget T660:=[[44.499965,36.567548,6.249631],[1.000000,0.000000,0.000000,0.000000],[0,0,-1,0],[9E+09,9E+09,9E+09,9E+09,9E+09,9E+09]];
    CONST robtarget T661:=[[44.499965,74.486666,6.249631],[1.000000,0.000000,0.000000,0.000000],[0,0,-1,0],[9E+09,9E+09,9E+09,9E+09,9E+09,9E+09]];
    CONST robtarget T662:=[[45.999971,75.305595,6.249631],[1.000000,0.000000,0.000000,0.000000],[0,0,-1,0],[9E+09,9E+09,9E+09,9E+09,9E+09,9E+09]];
    CONST robtarget T663:=[[45.999971,36.214678,6.249631],[1.000000,0.000000,0.000000,0.000000],[0,0,-1,0],[9E+09,9E+09,9E+09,9E+09,9E+09,9E+09]];
    CONST robtarget T664:=[[47.499977,35.829098,6.249631],[1.000000,0.000000,0.000000,0.000000],[0,0,-1,0],[9E+09,9E+09,9E+09,9E+09,9E+09,9E+09]];
    CONST robtarget T665:=[[47.499977,75.849984,6.249631],[1.000000,0.000000,0.000000,0.000000],[0,0,-1,0],[9E+09,9E+09,9E+09,9E+09,9E+09,9E+09]];
    CONST robtarget T666:=[[48.999983,76.089977,6.249631],[1.000000,0.000000,0.000000,0.000000],[0,0,-1,0],[9E+09,9E+09,9E+09,9E+09,9E+09,9E+09]];
    CONST robtarget T667:=[[48.999983,35.612525,6.249631],[1.000000,0.000000,0.000000,0.000000],[0,0,-1,0],[9E+09,9E+09,9E+09,9E+09,9E+09,9E+09]];
    CONST robtarget T668:=[[50.499989,35.473840,6.249631],[1.000000,0.000000,0.000000,0.000000],[0,0,-1,0],[9E+09,9E+09,9E+09,9E+09,9E+09,9E+09]];
    CONST robtarget T669:=[[50.499989,76.264329,6.249631],[1.000000,0.000000,0.000000,0.000000],[0,0,-1,0],[9E+09,9E+09,9E+09,9E+09,9E+09,9E+09]];
    CONST robtarget T670:=[[51.999995,76.384788,6.249631],[1.000000,0.000000,0.000000,0.000000],[0,0,-1,0],[9E+09,9E+09,9E+09,9E+09,9E+09,9E+09]];
    CONST robtarget T671:=[[51.999995,35.406248,6.249631],[1.000000,0.000000,0.000000,0.000000],[0,0,-1,0],[9E+09,9E+09,9E+09,9E+09,9E+09,9E+09]];
    CONST robtarget T672:=[[53.500001,35.366345,6.249631],[1.000000,0.000000,0.000000,0.000000],[0,0,-1,0],[9E+09,9E+09,9E+09,9E+09,9E+09,9E+09]];
    CONST robtarget T673:=[[53.500001,76.537077,6.249631],[1.000000,0.000000,0.000000,0.000000],[0,0,-1,0],[9E+09,9E+09,9E+09,9E+09,9E+09,9E+09]];
    CONST robtarget T674:=[[55.000007,76.638151,6.249631],[1.000000,0.000000,0.000000,0.000000],[0,0,-1,0],[9E+09,9E+09,9E+09,9E+09,9E+09,9E+09]];
    CONST robtarget T675:=[[55.000007,35.370600,6.249631],[1.000000,0.000000,0.000000,0.000000],[0,0,-1,0],[9E+09,9E+09,9E+09,9E+09,9E+09,9E+09]];
    CONST robtarget T676:=[[56.500013,35.366345,6.249631],[1.000000,0.000000,0.000000,0.000000],[0,0,-1,0],[9E+09,9E+09,9E+09,9E+09,9E+09,9E+09]];
